C01854=1122.207,107.838,-57.449,-179.830,8.137,149.506
C01855=1122.202,108.087,-57.468,-179.828,8.140,149.507
C01856=1122.197,108.336,-57.487,-179.826,8.144,149.507
C01857=1122.193,108.586,-57.507,-179.823,8.148,149.507
C01858=1122.187,108.834,-57.526,-179.821,8.151,149.507
C01859=1122.183,109.084,-57.546,-179.818,8.156,149.507
C01860=1122.179,109.333,-57.565,-179.817,8.160,149.508
C01861=1122.173,109.582,-57.584,-179.815,8.163,149.508
C01862=1122.168,109.832,-57.604,-179.812,8.167,149.508
C01863=1122.163,110.081,-57.623,-179.810,8.171,149.509
C01864=1122.158,110.330,-57.642,-179.807,8.175,149.509
C01865=1122.154,110.579,-57.662,-179.805,8.179,149.509
C01866=1122.149,110.828,-57.681,-179.802,8.183,149.509
C01867=1122.144,111.078,-57.700,-179.800,8.186,149.509
C01868=1122.140,111.327,-57.720,-179.798,8.190,149.510
C01869=1122.135,111.576,-57.740,-179.796,8.193,149.510
C01870=1122.130,111.825,-57.760,-179.795,8.196,149.510
C01871=1122.125,112.075,-57.779,-179.793,8.200,149.511
C01872=1122.120,112.323,-57.798,-179.791,8.203,149.511
C01873=1122.116,112.573,-57.818,-179.789,8.207,149.511
C01874=1122.111,112.822,-57.838,-179.787,8.210,149.511
C01875=1122.106,113.071,-57.857,-179.786,8.214,149.512
C01876=1122.101,113.320,-57.877,-179.783,8.218,149.512
C01877=1122.096,113.570,-57.897,-179.781,8.221,149.512
C01878=1122.091,113.818,-57.917,-179.779,8.225,149.512
C01879=1122.087,114.068,-57.936,-179.778,8.228,149.513
C01880=1122.082,114.317,-57.956,-179.776,8.231,149.513
C01881=1122.077,114.567,-57.976,-179.774,8.235,149.513
C01882=1122.072,114.815,-57.996,-179.772,8.238,149.513
C01883=1122.067,115.065,-58.015,-179.771,8.242,149.514
C01884=1122.063,115.314,-58.035,-179.768,8.246,149.514
C01885=1122.058,115.563,-58.055,-179.766,8.249,149.514
C01886=1122.053,115.812,-58.075,-179.765,8.252,149.515
C01887=1122.048,116.062,-58.094,-179.763,8.256,149.515
C01888=1122.045,116.275,-58.111,-179.762,8.259,149.515
C01889=1122.041,116.490,-58.128,-179.760,8.262,149.515
C01890=1122.036,116.704,-58.146,-179.758,8.265,149.516
C01891=1122.032,116.919,-58.163,-179.757,8.268,149.516
C01892=1122.028,117.133,-58.180,-179.755,8.271,149.516
C01893=1122.024,117.347,-58.197,-179.753,8.274,149.516
C01894=1122.020,117.562,-58.214,-179.752,8.277,149.517
C01895=1122.015,117.776,-58.231,-179.751,8.279,149.517
C01896=1122.011,118.026,-58.251,-179.749,8.283,149.517
C01897=1122.006,118.275,-58.271,-179.746,8.286,149.517
C01898=1122.001,118.524,-58.291,-179.745,8.290,149.518
C01899=1121.996,118.773,-58.311,-179.743,8.294,149.518
C01900=1121.992,119.022,-58.331,-179.741,8.296,149.518
C01901=1121.987,119.271,-58.351,-179.739,8.300,149.518
C01902=1121.983,119.521,-58.371,-179.738,8.304,149.519
C01903=1121.978,119.770,-58.391,-179.736,8.307,149.519
C01904=1121.973,120.019,-58.411,-179.734,8.310,149.519
C01905=1121.968,120.267,-58.431,-179.732,8.313,149.519
C01906=1121.963,120.517,-58.452,-179.730,8.317,149.520
C01907=1121.958,120.766,-58.471,-179.728,8.321,149.520
C01908=1121.954,121.015,-58.492,-179.727,8.324,149.520
C01909=1121.949,121.265,-58.511,-179.725,8.327,149.520
C01910=1121.945,121.514,-58.532,-179.723,8.331,149.521
C01911=1121.940,121.763,-58.552,-179.721,8.334,149.521
C01912=1121.935,122.012,-58.571,-179.720,8.337,149.521
C01913=1121.930,122.261,-58.592,-179.718,8.341,149.522
C01914=1121.925,122.510,-58.612,-179.716,8.344,149.522
C01915=1121.921,122.759,-58.632,-179.714,8.348,149.522
C01916=1121.916,123.008,-58.653,-179.713,8.351,149.522
C01917=1121.912,123.257,-58.673,-179.711,8.354,149.523
C01918=1121.906,123.507,-58.693,-179.708,8.358,149.523
C01919=1121.902,123.756,-58.714,-179.706,8.361,149.523
C01920=1121.897,124.005,-58.734,-179.705,8.364,149.523
C01921=1121.893,124.255,-58.754,-179.703,8.368,149.524
C01922=1121.887,124.504,-58.775,-179.701,8.371,149.524
C01923=1121.882,124.752,-58.795,-179.700,8.374,149.524
C01924=1121.878,125.001,-58.815,-179.698,8.377,149.524
C01925=1121.873,125.251,-58.835,-179.696,8.381,149.525
C01926=1121.868,125.500,-58.856,-179.695,8.384,149.525
C01927=1121.864,125.749,-58.876,-179.693,8.388,149.525
C01928=1121.859,125.998,-58.897,-179.691,8.391,149.526
C01929=1121.855,126.247,-58.917,-179.689,8.395,149.526
C01930=1121.850,126.496,-58.938,-179.687,8.398,149.526
C01931=1121.845,126.746,-58.958,-179.685,8.401,149.526
C01932=1121.840,126.994,-58.978,-179.683,8.405,149.527
C01933=1121.835,127.244,-58.999,-179.682,8.407,149.527
C01934=1121.831,127.493,-59.019,-179.680,8.411,149.527
C01935=1121.826,127.742,-59.040,-179.678,8.415,149.528
C01936=1121.821,127.991,-59.061,-179.677,8.417,149.528
C01937=1121.817,128.240,-59.081,-179.675,8.421,149.528
C01938=1121.812,128.489,-59.101,-179.673,8.425,149.528
C01939=1121.807,128.739,-59.122,-179.672,8.428,149.529
C01940=1121.802,128.988,-59.142,-179.670,8.431,149.529
C01941=1121.797,129.237,-59.163,-179.668,8.435,149.529
C01942=1121.793,129.486,-59.183,-179.666,8.438,149.530
C01943=1121.788,129.735,-59.204,-179.664,8.441,149.530
C01944=1121.784,129.950,-59.222,-179.663,8.444,149.530
C01945=1121.780,130.163,-59.239,-179.662,8.447,149.530
C01946=1121.776,130.378,-59.257,-179.660,8.449,149.530
C01947=1121.772,130.592,-59.275,-179.659,8.452,149.531
C01948=1121.768,130.806,-59.292,-179.657,8.456,149.531
C01949=1121.764,131.021,-59.311,-179.656,8.459,149.531
C01950=1121.759,131.235,-59.328,-179.654,8.461,149.532
C01951=1121.756,131.449,-59.346,-179.653,8.464,149.532
C01952=1121.751,131.699,-59.367,-179.651,8.467,149.532
C01953=1121.746,131.947,-59.387,-179.650,8.471,149.532
C01954=1121.741,132.196,-59.409,-179.648,8.474,149.533
C01955=1121.737,132.445,-59.429,-179.646,8.477,149.533
C01956=1121.732,132.694,-59.450,-179.644,8.480,149.533
C01957=1121.727,132.943,-59.471,-179.642,8.484,149.534
C01958=1121.722,133.193,-59.492,-179.641,8.487,149.534
C01959=1121.718,133.441,-59.512,-179.639,8.490,149.534
C01960=1121.713,133.691,-59.533,-179.638,8.493,149.534
C01961=1121.709,133.940,-59.554,-179.636,8.497,149.535
C01962=1121.704,134.189,-59.575,-179.634,8.500,149.535
C01963=1121.699,134.438,-59.596,-179.633,8.504,149.535
C01964=1121.694,134.687,-59.617,-179.631,8.507,149.536
C01965=1121.690,134.936,-59.637,-179.629,8.510,149.536
C01966=1121.685,135.185,-59.658,-179.628,8.514,149.536
C01967=1121.680,135.434,-59.679,-179.625,8.517,149.536
C01968=1121.675,135.683,-59.700,-179.624,8.520,149.537
C01969=1121.671,135.933,-59.721,-179.622,8.524,149.537
C01970=1121.666,136.182,-59.742,-179.621,8.526,149.537
C01971=1121.661,136.431,-59.764,-179.619,8.530,149.538
C01972=1121.657,136.680,-59.784,-179.617,8.534,149.538
C01973=1121.652,136.929,-59.805,-179.616,8.536,149.538
C01974=1121.647,137.178,-59.826,-179.614,8.540,149.539
C01975=1121.643,137.426,-59.847,-179.613,8.543,149.539
C01976=1121.638,137.676,-59.868,-179.611,8.547,149.539
C01977=1121.633,137.926,-59.889,-179.609,8.550,149.540
C01978=1121.629,138.174,-59.910,-179.608,8.554,149.540
C01979=1121.623,138.423,-59.931,-179.606,8.557,149.540
C01980=1121.619,138.672,-59.952,-179.604,8.560,149.540
C01981=1121.615,138.921,-59.974,-179.603,8.564,149.541
C01982=1121.610,139.171,-59.995,-179.601,8.566,149.541
C01983=1121.605,139.419,-60.016,-179.600,8.570,149.542
C01984=1121.600,139.668,-60.037,-179.598,8.574,149.542
C01985=1121.595,139.918,-60.058,-179.597,8.577,149.542
C01986=1121.591,140.167,-60.080,-179.595,8.580,149.542
C01987=1121.586,140.416,-60.100,-179.594,8.583,149.543
C01988=1121.582,140.665,-60.122,-179.592,8.587,149.543
C01989=1121.576,140.914,-60.143,-179.591,8.590,149.544
C01990=1121.573,141.163,-60.164,-179.588,8.593,149.544
C01991=1121.568,141.412,-60.185,-179.587,8.596,149.544
C01992=1121.563,141.661,-60.207,-179.585,8.600,149.544
C01993=1121.558,141.910,-60.228,-179.584,8.604,149.545
C01994=1121.554,142.159,-60.249,-179.582,8.607,149.545
C01995=1121.549,142.408,-60.270,-179.581,8.610,149.546
C01996=1121.544,142.657,-60.292,-179.579,8.613,149.546
C01997=1121.539,142.906,-60.313,-179.578,8.617,149.546
C01998=1121.535,143.155,-60.334,-179.576,8.620,149.546
C01999=1121.530,143.404,-60.355,-179.574,8.624,149.547
C02000=1121.526,143.619,-60.374,-179.573,8.626,149.547
C02001=1121.522,143.832,-60.392,-179.572,8.629,149.548
C02002=1121.518,144.047,-60.411,-179.571,8.632,149.548
C02003=1121.514,144.261,-60.429,-179.569,8.635,149.548
C02004=1121.510,144.475,-60.448,-179.568,8.638,149.548
C02005=1121.506,144.690,-60.466,-179.567,8.641,149.549
C02006=1121.502,144.903,-60.484,-179.565,8.643,149.549
C02007=1121.497,145.118,-60.503,-179.564,8.646,149.549
C02008=1121.493,145.366,-60.524,-179.561,8.651,149.550
C02009=1121.489,145.616,-60.546,-179.559,8.654,149.550
C02010=1121.484,145.865,-60.567,-179.557,8.658,149.550
C02011=1121.479,146.114,-60.588,-179.555,8.662,149.550
C02012=1121.475,146.363,-60.610,-179.552,8.666,149.550
C02013=1121.469,146.612,-60.631,-179.549,8.669,149.551
C02014=1121.464,146.861,-60.653,-179.547,8.674,149.551
C02015=1121.460,147.110,-60.675,-179.545,8.677,149.551
C02016=1121.455,147.359,-60.697,-179.542,8.681,149.551
C02017=1121.451,147.609,-60.718,-179.540,8.685,149.551
C02018=1121.447,147.857,-60.739,-179.538,8.688,149.552
C02019=1121.442,148.106,-60.761,-179.535,8.693,149.552
C02020=1121.438,148.355,-60.783,-179.533,8.696,149.552
C02021=1121.433,148.604,-60.805,-179.530,8.700,149.552
C02022=1121.427,148.853,-60.826,-179.528,8.703,149.552
C02023=1121.423,149.102,-60.848,-179.526,8.707,149.553
C02024=1121.418,149.351,-60.869,-179.523,8.711,149.553
C02025=1121.414,149.600,-60.891,-179.520,8.714,149.553
C02026=1121.409,149.849,-60.913,-179.518,8.719,149.553
C02027=1121.404,150.098,-60.935,-179.516,8.722,149.553
C02028=1121.400,150.347,-60.957,-179.513,8.726,149.554
C02029=1121.394,150.596,-60.979,-179.510,8.729,149.554
C02030=1121.390,150.845,-61.001,-179.508,8.733,149.554
C02031=1121.385,151.094,-61.023,-179.506,8.736,149.554
C02032=1121.381,151.343,-61.045,-179.504,8.740,149.554
C02033=1121.376,151.592,-61.067,-179.501,8.744,149.554
C02034=1121.372,151.842,-61.088,-179.499,8.747,149.555
C02035=1121.367,152.090,-61.110,-179.497,8.751,149.555
C02036=1121.362,152.338,-61.132,-179.494,8.755,149.555
C02037=1121.358,152.588,-61.154,-179.492,8.758,149.555
C02038=1121.353,152.836,-61.176,-179.489,8.762,149.555
C02039=1121.348,153.086,-61.198,-179.487,8.765,149.555
C02040=1121.343,153.335,-61.220,-179.484,8.769,149.556
C02041=1121.339,153.584,-61.242,-179.482,8.772,149.556
C02042=1121.334,153.833,-61.264,-179.480,8.776,149.556
C02043=1121.330,154.082,-61.286,-179.478,8.779,149.556
C02044=1121.325,154.331,-61.307,-179.475,8.782,149.556
C02045=1121.320,154.580,-61.330,-179.472,8.786,149.556
C02046=1121.316,154.830,-61.352,-179.470,8.790,149.556
C02047=1121.311,155.078,-61.375,-179.468,8.793,149.557
C02048=1121.307,155.327,-61.397,-179.465,8.796,149.557
C02049=1121.302,155.576,-61.418,-179.463,8.800,149.557
C02050=1121.297,155.825,-61.441,-179.461,8.803,149.557
C02051=1121.292,156.074,-61.463,-179.458,8.807,149.557
C02052=1121.288,156.323,-61.485,-179.455,8.810,149.557
C02053=1121.283,156.571,-61.507,-179.453,8.814,149.557
C02054=1121.278,156.821,-61.530,-179.451,8.817,149.558
C02055=1121.274,157.070,-61.552,-179.449,8.820,149.558
C02056=1121.270,157.284,-61.572,-179.446,8.823,149.558
C02057=1121.266,157.498,-61.591,-179.445,8.826,149.558
C02058=1121.262,157.712,-61.610,-179.442,8.829,149.558
C02059=1121.258,157.927,-61.629,-179.441,8.832,149.558
C02060=1121.254,158.141,-61.648,-179.438,8.835,149.558
C02061=1121.250,158.355,-61.667,-179.436,8.837,149.558
C02062=1121.247,158.568,-61.686,-179.434,8.841,149.559
C02063=1121.243,158.782,-61.705,-179.432,8.843,149.559
C02064=1121.237,159.031,-61.728,-179.430,8.847,149.559
C02065=1121.233,159.280,-61.750,-179.428,8.850,149.559
C02066=1121.229,159.529,-61.772,-179.426,8.853,149.559
C02067=1121.223,159.778,-61.795,-179.423,8.856,149.559
C02068=1121.219,160.027,-61.817,-179.421,8.859,149.559
C02069=1121.214,160.277,-61.840,-179.418,8.864,149.559
C02070=1121.210,160.525,-61.862,-179.415,8.867,149.559
C02071=1121.205,160.774,-61.885,-179.413,8.870,149.560
C02072=1121.201,161.023,-61.908,-179.411,8.873,149.560
C02073=1121.196,161.272,-61.930,-179.408,8.876,149.560
C02074=1121.191,161.521,-61.953,-179.406,8.880,149.560
C02075=1121.187,161.770,-61.975,-179.404,8.882,149.560
C02076=1121.182,162.018,-61.997,-179.402,8.885,149.560
C02077=1121.177,162.268,-62.020,-179.400,8.889,149.560
C02078=1121.173,162.516,-62.043,-179.397,8.892,149.560
C02079=1121.168,162.765,-62.065,-179.395,8.895,149.561
C02080=1121.164,163.014,-62.088,-179.393,8.899,149.561
C02081=1121.159,163.263,-62.111,-179.390,8.902,149.561
C02082=1121.155,163.513,-62.133,-179.388,8.905,149.561
C02083=1121.149,163.761,-62.156,-179.385,8.908,149.561
C02084=1121.145,164.010,-62.178,-179.383,8.911,149.561
C02085=1121.141,164.259,-62.202,-179.381,8.915,149.561
C02086=1121.137,164.508,-62.224,-179.378,8.918,149.561
C02087=1121.131,164.757,-62.247,-179.376,8.921,149.561
C02088=1121.127,165.006,-62.269,-179.374,8.925,149.561
C02089=1121.122,165.255,-62.293,-179.371,8.928,149.561
C02090=1121.118,165.504,-62.315,-179.369,8.930,149.562
C02091=1121.113,165.752,-62.338,-179.367,8.933,149.562
C02092=1121.108,166.001,-62.361,-179.365,8.937,149.562
C02093=1121.104,166.250,-62.384,-179.362,8.940,149.562
C02094=1121.099,166.500,-62.407,-179.360,8.943,149.562
C02095=1121.095,166.748,-62.429,-179.357,8.946,149.562
C02096=1121.090,166.997,-62.452,-179.355,8.949,149.562
C02097=1121.085,167.246,-62.476,-179.353,8.952,149.562
C02098=1121.081,167.495,-62.498,-179.351,8.955,149.562
C02099=1121.076,167.744,-62.521,-179.348,8.958,149.562
C02100=1121.071,167.993,-62.544,-179.346,8.961,149.562
C02101=1121.067,168.241,-62.567,-179.344,8.965,149.563
C02102=1121.062,168.490,-62.590,-179.341,8.968,149.563
C02103=1121.057,168.739,-62.614,-179.339,8.970,149.563
C02104=1121.053,168.988,-62.636,-179.337,8.974,149.563
C02105=1121.048,169.238,-62.659,-179.335,8.977,149.563
C02106=1121.044,169.487,-62.682,-179.332,8.980,149.563
C02107=1121.039,169.735,-62.705,-179.330,8.983,149.563
C02108=1121.035,169.984,-62.728,-179.328,8.986,149.563
C02109=1121.030,170.233,-62.751,-179.326,8.989,149.563
C02110=1121.026,170.482,-62.774,-179.323,8.992,149.563
C02111=1121.021,170.731,-62.798,-179.321,8.996,149.564
C02112=1121.017,170.944,-62.817,-179.319,8.998,149.564
C02113=1121.013,171.158,-62.838,-179.317,9.000,149.564
C02114=1121.009,171.373,-62.857,-179.315,9.003,149.564
C02115=1121.006,171.586,-62.877,-179.313,9.006,149.564
C02116=1121.001,171.800,-62.897,-179.312,9.008,149.564
C02117=1120.997,172.014,-62.917,-179.310,9.011,149.564
C02118=1120.994,172.229,-62.937,-179.308,9.013,149.564
C02119=1120.989,172.443,-62.957,-179.306,9.016,149.564
C02120=1120.985,172.692,-62.980,-179.304,9.019,149.564
C02121=1120.981,172.940,-63.003,-179.301,9.022,149.564
C02122=1120.976,173.189,-63.027,-179.300,9.025,149.565
C02123=1120.971,173.437,-63.050,-179.297,9.028,149.565
C02124=1120.966,173.686,-63.074,-179.295,9.031,149.565
C02125=1120.962,173.935,-63.097,-179.292,9.034,149.565
C02126=1120.957,174.184,-63.120,-179.291,9.037,149.565
C02127=1120.953,174.433,-63.143,-179.288,9.040,149.565
C02128=1120.948,174.682,-63.167,-179.286,9.043,149.565
C02129=1120.943,174.931,-63.190,-179.284,9.046,149.565
C02130=1120.939,175.179,-63.214,-179.282,9.049,149.565
C02131=1120.934,175.428,-63.237,-179.279,9.052,149.565
C02132=1120.930,175.677,-63.261,-179.278,9.055,149.566
C02133=1120.925,175.927,-63.284,-179.275,9.058,149.566
C02134=1120.921,176.175,-63.307,-179.273,9.061,149.566
C02135=1120.917,176.424,-63.331,-179.271,9.063,149.566
C02136=1120.912,176.673,-63.354,-179.269,9.067,149.566
C02137=1120.907,176.922,-63.378,-179.266,9.070,149.566
C02138=1120.903,177.171,-63.401,-179.264,9.072,149.566
C02139=1120.898,177.419,-63.425,-179.262,9.075,149.566
C02140=1120.893,177.668,-63.448,-179.260,9.079,149.566
C02141=1120.889,177.917,-63.472,-179.258,9.081,149.566
C02142=1120.884,178.166,-63.496,-179.256,9.084,149.567
C02143=1120.880,178.415,-63.519,-179.254,9.087,149.567
C02144=1120.875,178.664,-63.543,-179.252,9.090,149.567
C02145=1120.871,178.912,-63.567,-179.249,9.093,149.567
C02146=1120.866,179.161,-63.590,-179.247,9.096,149.567
C02147=1120.861,179.410,-63.613,-179.245,9.099,149.567
C02148=1120.857,179.659,-63.637,-179.242,9.103,149.567
C02149=1120.852,179.908,-63.661,-179.239,9.106,149.567
C02150=1120.848,180.157,-63.684,-179.237,9.109,149.567
C02151=1120.844,180.406,-63.709,-179.234,9.112,149.567
C02152=1120.839,180.655,-63.732,-179.231,9.116,149.567
C02153=1120.834,180.903,-63.756,-179.228,9.119,149.567
C02154=1120.830,181.152,-63.779,-179.225,9.122,149.567
C02155=1120.825,181.401,-63.803,-179.223,9.125,149.567
C02156=1120.821,181.650,-63.827,-179.220,9.128,149.567
C02157=1120.816,181.898,-63.851,-179.218,9.131,149.567
C02158=1120.812,182.147,-63.874,-179.215,9.135,149.567
C02159=1120.807,182.396,-63.898,-179.212,9.138,149.567
C02160=1120.802,182.646,-63.923,-179.209,9.141,149.567
C02161=1120.798,182.894,-63.947,-179.207,9.144,149.567
C02162=1120.793,183.143,-63.970,-179.204,9.147,149.567
C02163=1120.789,183.391,-63.994,-179.202,9.150,149.567
C02164=1120.784,183.640,-64.018,-179.199,9.153,149.567
C02165=1120.780,183.889,-64.042,-179.197,9.156,149.567
C02166=1120.775,184.137,-64.066,-179.194,9.159,149.567
C02167=1120.771,184.387,-64.091,-179.191,9.162,149.567
C02168=1120.767,184.600,-64.110,-179.189,9.164,149.567
C02169=1120.763,184.814,-64.131,-179.187,9.167,149.567
C02170=1120.759,185.028,-64.152,-179.185,9.170,149.567
C02171=1120.755,185.242,-64.172,-179.183,9.172,149.567
C02172=1120.751,185.456,-64.193,-179.181,9.175,149.567
C02173=1120.747,185.670,-64.214,-179.179,9.177,149.567
C02174=1120.744,185.884,-64.234,-179.177,9.180,149.568
C02175=1120.740,186.097,-64.255,-179.175,9.182,149.568
C02176=1120.735,186.346,-64.279,-179.172,9.185,149.567
C02177=1120.730,186.596,-64.304,-179.170,9.187,149.567
C02178=1120.726,186.844,-64.328,-179.167,9.191,149.567
C02179=1120.722,187.092,-64.352,-179.165,9.194,149.568
C02180=1120.717,187.341,-64.376,-179.162,9.197,149.568
C02181=1120.712,187.591,-64.400,-179.160,9.199,149.568
C02182=1120.708,187.839,-64.424,-179.158,9.202,149.568
C02183=1120.704,188.088,-64.448,-179.155,9.205,149.568
C02184=1120.698,188.336,-64.473,-179.153,9.208,149.568
C02185=1120.694,188.585,-64.497,-179.151,9.211,149.568
C02186=1120.690,188.834,-64.522,-179.149,9.213,149.568
C02187=1120.685,189.083,-64.546,-179.146,9.216,149.568
C02188=1120.680,189.332,-64.570,-179.144,9.219,149.568
C02189=1120.676,189.580,-64.594,-179.142,9.222,149.568
C02190=1120.672,189.829,-64.619,-179.140,9.225,149.568
C02191=1120.667,190.078,-64.643,-179.138,9.227,149.568
C02192=1120.662,190.327,-64.667,-179.135,9.230,149.568
C02193=1120.658,190.576,-64.692,-179.133,9.232,149.568
C02194=1120.654,190.824,-64.716,-179.131,9.236,149.568
C02195=1120.649,191.073,-64.741,-179.129,9.238,149.568
C02196=1120.644,191.321,-64.765,-179.127,9.241,149.568
C02197=1120.640,191.571,-64.790,-179.125,9.244,149.568
C02198=1120.635,191.819,-64.814,-179.123,9.246,149.569
C02199=1120.631,192.067,-64.838,-179.120,9.249,149.569
C02200=1120.626,192.317,-64.863,-179.119,9.252,149.569
C02201=1120.622,192.565,-64.887,-179.117,9.254,149.569
C02202=1120.617,192.814,-64.912,-179.115,9.257,149.569
C02203=1120.613,193.063,-64.936,-179.113,9.260,149.569
C02204=1120.608,193.312,-64.961,-179.111,9.262,149.569
C02205=1120.604,193.560,-64.985,-179.109,9.265,149.569
C02206=1120.599,193.810,-65.010,-179.107,9.268,149.569
C02207=1120.595,194.058,-65.034,-179.105,9.270,149.569
C02208=1120.590,194.307,-65.059,-179.103,9.273,149.570
C02209=1120.586,194.556,-65.083,-179.101,9.276,149.570
C02210=1120.581,194.805,-65.108,-179.099,9.279,149.570
C02211=1120.577,195.052,-65.133,-179.097,9.281,149.570
C02212=1120.572,195.302,-65.158,-179.096,9.284,149.570
C02213=1120.568,195.550,-65.182,-179.094,9.286,149.570
C02214=1120.563,195.800,-65.207,-179.092,9.289,149.570
C02215=1120.559,196.048,-65.231,-179.090,9.292,149.570
C02216=1120.554,196.297,-65.255,-179.089,9.295,149.571
C02217=1120.550,196.545,-65.281,-179.086,9.298,149.571
C02218=1120.545,196.794,-65.305,-179.083,9.301,149.571
C02219=1120.541,197.043,-65.330,-179.079,9.305,149.570
C02220=1120.536,197.292,-65.354,-179.076,9.309,149.570
C02221=1120.532,197.540,-65.379,-179.072,9.312,149.570
C02222=1120.527,197.789,-65.404,-179.069,9.315,149.570
C02223=1120.522,198.038,-65.429,-179.066,9.319,149.570
C02224=1120.519,198.252,-65.450,-179.063,9.321,149.570
C02225=1120.515,198.466,-65.472,-179.061,9.325,149.570
C02226=1120.511,198.679,-65.493,-179.058,9.327,149.570
C02227=1120.507,198.893,-65.514,-179.055,9.330,149.570
C02228=1120.504,199.107,-65.536,-179.052,9.333,149.570
C02229=1120.499,199.320,-65.557,-179.049,9.336,149.570
C02230=1120.496,199.534,-65.578,-179.046,9.339,149.570
C02231=1120.492,199.748,-65.600,-179.044,9.342,149.570
C02232=1120.487,199.997,-65.625,-179.041,9.344,149.570
C02233=1120.484,200.245,-65.650,-179.037,9.348,149.569
C02234=1120.478,200.494,-65.674,-179.034,9.351,149.569
C02235=1120.474,200.743,-65.700,-179.031,9.355,149.569
C02236=1120.469,200.992,-65.725,-179.028,9.357,149.569
C02237=1120.466,201.240,-65.750,-179.025,9.360,149.569
C02238=1120.460,201.489,-65.775,-179.022,9.364,149.569
C02239=1120.456,201.738,-65.800,-179.019,9.366,149.569
C02240=1120.451,201.986,-65.825,-179.016,9.369,149.569
C02241=1120.448,202.235,-65.850,-179.013,9.373,149.569
C02242=1120.443,202.484,-65.875,-179.010,9.376,149.569
C02243=1120.438,202.732,-65.901,-179.007,9.378,149.568
C02244=1120.433,202.980,-65.926,-179.004,9.381,149.568
C02245=1120.430,203.230,-65.950,-179.001,9.385,149.568
C02246=1120.425,203.478,-65.976,-178.998,9.388,149.568
C02247=1120.420,203.727,-66.001,-178.995,9.391,149.568
C02248=1120.416,203.976,-66.027,-178.992,9.393,149.568
C02249=1120.411,204.224,-66.052,-178.989,9.396,149.568
C02250=1120.407,204.473,-66.077,-178.986,9.399,149.568
C02251=1120.403,204.722,-66.103,-178.983,9.402,149.568
C02252=1120.398,204.970,-66.128,-178.980,9.405,149.567
C02253=1120.394,205.219,-66.153,-178.977,9.408,149.567
C02254=1120.389,205.468,-66.178,-178.974,9.411,149.567
C02255=1120.385,205.716,-66.204,-178.971,9.414,149.567
C02256=1120.381,205.965,-66.230,-178.968,9.417,149.567
C02257=1120.375,206.214,-66.254,-178.966,9.420,149.567
C02258=1120.371,206.463,-66.280,-178.963,9.423,149.567
C02259=1120.366,206.711,-66.305,-178.961,9.425,149.567
C02260=1120.362,206.960,-66.331,-178.958,9.428,149.567
C02261=1120.358,207.208,-66.357,-178.955,9.430,149.567
C02262=1120.353,207.457,-66.382,-178.952,9.433,149.567
C02263=1120.349,207.706,-66.407,-178.950,9.436,149.567
C02264=1120.344,207.955,-66.433,-178.947,9.439,149.567
C02265=1120.340,208.203,-66.458,-178.944,9.442,149.567
C02266=1120.335,208.452,-66.484,-178.941,9.445,149.566
C02267=1120.331,208.700,-66.510,-178.939,9.448,149.566
C02268=1120.326,208.949,-66.535,-178.936,9.450,149.566
C02269=1120.322,209.197,-66.561,-178.934,9.453,149.566
C02270=1120.318,209.446,-66.587,-178.931,9.456,149.566
C02271=1120.314,209.695,-66.613,-178.928,9.459,149.566
C02272=1120.309,209.943,-66.638,-178.926,9.462,149.566
C02273=1120.305,210.192,-66.664,-178.923,9.464,149.566
C02274=1120.300,210.441,-66.689,-178.921,9.467,149.566
C02275=1120.296,210.689,-66.715,-178.918,9.470,149.566
C02276=1120.291,210.938,-66.741,-178.916,9.473,149.566
C02277=1120.287,211.186,-66.766,-178.914,9.475,149.566
C02278=1120.282,211.436,-66.793,-178.911,9.478,149.566
C02279=1120.277,211.684,-66.818,-178.909,9.481,149.566
C02280=1120.274,211.898,-66.840,-178.907,9.484,149.566
C02281=1120.270,212.111,-66.862,-178.905,9.486,149.566
C02282=1120.266,212.325,-66.885,-178.903,9.488,149.566
C02283=1120.263,212.539,-66.906,-178.901,9.491,149.567
C02284=1120.259,212.752,-66.929,-178.898,9.494,149.567
C02285=1120.255,212.966,-66.951,-178.897,9.496,149.567
C02286=1120.251,213.180,-66.973,-178.895,9.499,149.567
C02287=1120.248,213.393,-66.995,-178.893,9.501,149.567
C02288=1120.242,213.642,-67.021,-178.891,9.504,149.567
C02289=1120.238,213.890,-67.047,-178.889,9.507,149.567
C02290=1120.234,214.139,-67.073,-178.887,9.509,149.567
C02291=1120.230,214.387,-67.099,-178.885,9.513,149.567
C02292=1120.226,214.636,-67.125,-178.883,9.515,149.567
C02293=1120.221,214.884,-67.150,-178.881,9.518,149.568
C02294=1120.216,215.133,-67.177,-178.879,9.521,149.568
C02295=1120.212,215.382,-67.202,-178.876,9.524,149.568
C02296=1120.208,215.630,-67.229,-178.875,9.526,149.568
C02297=1120.203,215.879,-67.255,-178.872,9.530,149.568
C02298=1120.198,216.128,-67.281,-178.870,9.532,149.568
C02299=1120.194,216.376,-67.306,-178.868,9.535,149.568
C02300=1120.190,216.625,-67.333,-178.866,9.538,149.568
C02301=1120.185,216.873,-67.359,-178.864,9.541,149.568
C02302=1120.181,217.122,-67.385,-178.862,9.544,149.569
C02303=1120.177,217.371,-67.411,-178.859,9.547,149.569
C02304=1120.170,217.694,-67.445,-178.857,9.551,149.569
C02305=1120.165,218.019,-67.479,-178.854,9.555,149.569
C02306=1120.159,218.343,-67.513,-178.851,9.559,149.569
C02307=1120.154,218.667,-67.548,-178.848,9.563,149.569
C02308=1120.149,218.915,-67.573,-178.845,9.566,149.569
C02309=1120.144,219.164,-67.600,-178.843,9.569,149.570
C02310=1120.140,219.412,-67.626,-178.841,9.572,149.570
C02311=1120.136,219.661,-67.651,-178.838,9.575,149.570
C02312=1120.131,219.910,-67.679,-178.836,9.578,149.570
C02313=1120.127,220.158,-67.704,-178.833,9.582,149.570
C02314=1120.122,220.407,-67.731,-178.831,9.584,149.570
C02315=1120.118,220.656,-67.757,-178.829,9.587,149.570
C02316=1120.114,220.904,-67.784,-178.826,9.590,149.570
C02317=1120.109,221.153,-67.810,-178.824,9.594,149.570
C02318=1120.105,221.401,-67.836,-178.821,9.597,149.570
C02319=1120.101,221.650,-67.863,-178.819,9.600,149.570
C02320=1120.096,221.898,-67.889,-178.816,9.603,149.571
C02321=1120.091,222.147,-67.915,-178.813,9.607,149.571
C02322=1120.087,222.395,-67.942,-178.811,9.610,149.571
C02323=1120.083,222.643,-67.968,-178.808,9.613,149.571
C02324=1120.078,222.892,-67.994,-178.805,9.616,149.571
C02325=1120.074,223.141,-68.021,-178.803,9.619,149.571
C02326=1120.069,223.390,-68.047,-178.800,9.622,149.571
C02327=1120.065,223.638,-68.074,-178.798,9.625,149.571
C02328=1120.061,223.886,-68.101,-178.794,9.629,149.571
C02329=1120.057,224.135,-68.127,-178.792,9.632,149.571
C02330=1120.052,224.384,-68.154,-178.789,9.635,149.571
C02331=1120.048,224.632,-68.180,-178.786,9.638,149.571
C02332=1120.043,224.880,-68.207,-178.784,9.641,149.571
C02333=1120.039,225.129,-68.233,-178.781,9.645,149.571
C02334=1120.034,225.378,-68.260,-178.778,9.648,149.571
C02335=1120.030,225.626,-68.287,-178.775,9.651,149.571
C02336=1120.024,225.979,-68.325,-178.772,9.655,149.571
C02337=1120.018,226.330,-68.363,-178.767,9.661,149.571
C02338=1120.012,226.682,-68.400,-178.762,9.665,149.571
C02339=1120.005,227.033,-68.438,-178.759,9.669,149.571
C02340=1120.002,227.281,-68.465,-178.756,9.672,149.571
C02341=1119.997,227.530,-68.491,-178.753,9.676,149.571
C02342=1119.992,227.779,-68.518,-178.750,9.679,149.571
C02343=1119.988,228.027,-68.544,-178.746,9.682,149.571
C02344=1119.983,228.275,-68.572,-178.743,9.685,149.571
C02345=1119.979,228.524,-68.599,-178.741,9.688,149.571
C02346=1119.975,228.773,-68.625,-178.737,9.692,149.571
C02347=1119.971,229.021,-68.652,-178.734,9.695,149.570
C02348=1119.966,229.270,-68.680,-178.731,9.698,149.571
C02349=1119.961,229.518,-68.707,-178.728,9.701,149.570
C02350=1119.957,229.766,-68.733,-178.724,9.705,149.570
C02351=1119.953,230.015,-68.760,-178.721,9.707,149.570
C02352=1119.948,230.263,-68.787,-178.718,9.711,149.570
C02353=1119.944,230.513,-68.815,-178.714,9.714,149.570
C02354=1119.940,230.761,-68.841,-178.711,9.717,149.570
C02355=1119.936,231.009,-68.868,-178.708,9.720,149.570
C02356=1119.931,231.258,-68.895,-178.705,9.723,149.570
C02357=1119.926,231.506,-68.922,-178.702,9.726,149.569
C02358=1119.922,231.754,-68.949,-178.699,9.729,149.569
C02359=1119.919,232.003,-68.977,-178.696,9.733,149.569
C02360=1119.914,232.251,-69.004,-178.693,9.736,149.569
C02361=1119.909,232.500,-69.031,-178.690,9.738,149.569
C02362=1119.905,232.748,-69.058,-178.687,9.741,149.569
C02363=1119.900,232.997,-69.085,-178.684,9.744,149.569
C02364=1119.896,233.246,-69.113,-178.681,9.747,149.569
C02365=1119.892,233.494,-69.140,-178.677,9.750,149.569
C02366=1119.888,233.742,-69.167,-178.674,9.753,149.569
C02367=1119.883,233.991,-69.194,-178.671,9.756,149.568
C02368=1119.879,234.239,-69.222,-178.669,9.758,149.568
C02369=1119.875,234.488,-69.249,-178.666,9.761,149.568
C02370=1119.870,234.736,-69.276,-178.663,9.764,149.568
C02371=1119.865,234.985,-69.303,-178.660,9.767,149.568
C02372=1119.861,235.233,-69.331,-178.657,9.770,149.568
C02373=1119.857,235.482,-69.358,-178.654,9.772,149.568
C02374=1119.852,235.730,-69.385,-178.652,9.774,149.568
C02375=1119.848,235.978,-69.413,-178.649,9.777,149.568
C02376=1119.844,236.227,-69.440,-178.646,9.780,149.567
C02377=1119.840,236.475,-69.468,-178.643,9.783,149.567
C02378=1119.835,236.723,-69.495,-178.640,9.785,149.567
C02379=1119.831,236.973,-69.522,-178.638,9.788,149.567
C02380=1119.827,237.221,-69.550,-178.635,9.791,149.567
C02381=1119.822,237.469,-69.577,-178.632,9.793,149.567
C02382=1119.819,237.718,-69.605,-178.629,9.796,149.567
C02383=1119.813,237.966,-69.633,-178.627,9.798,149.567
C02384=1119.809,238.214,-69.661,-178.625,9.801,149.567
C02385=1119.805,238.464,-69.688,-178.622,9.804,149.567
C02386=1119.801,238.711,-69.716,-178.619,9.806,149.567
C02387=1119.796,238.960,-69.743,-178.616,9.809,149.566
C02388=1119.793,239.174,-69.767,-178.614,9.811,149.566
C02389=1119.789,239.387,-69.790,-178.612,9.813,149.566
C02390=1119.785,239.600,-69.814,-178.610,9.815,149.566
C02391=1119.781,239.814,-69.838,-178.608,9.817,149.566
C02392=1119.778,240.027,-69.862,-178.606,9.820,149.566
C02393=1119.774,240.240,-69.885,-178.604,9.821,149.566
C02394=1119.771,240.453,-69.909,-178.602,9.824,149.566
C02395=1119.766,240.667,-69.933,-178.600,9.826,149.566
C02396=1119.762,240.915,-69.960,-178.598,9.828,149.566
C02397=1119.758,241.164,-69.989,-178.595,9.831,149.566
C02398=1119.754,241.412,-70.016,-178.593,9.833,149.566
C02399=1119.750,241.661,-70.044,-178.590,9.835,149.566
C02400=1119.745,241.909,-70.072,-178.588,9.838,149.566
C02401=1119.740,242.157,-70.100,-178.586,9.840,149.566
C02402=1119.736,242.406,-70.127,-178.584,9.843,149.566
C02403=1119.732,242.654,-70.155,-178.581,9.845,149.566
C02404=1119.728,242.903,-70.183,-178.579,9.848,149.566
C02405=1119.723,243.151,-70.210,-178.577,9.850,149.566
C02406=1119.719,243.399,-70.238,-178.575,9.852,149.566
C02407=1119.714,243.648,-70.267,-178.572,9.855,149.566
C02408=1119.710,243.896,-70.295,-178.570,9.857,149.566
C02409=1119.706,244.145,-70.322,-178.568,9.860,149.566
C02410=1119.702,244.393,-70.350,-178.566,9.862,149.566
C02411=1119.698,244.641,-70.378,-178.565,9.864,149.566
C02412=1119.693,244.890,-70.406,-178.563,9.867,149.566
C02413=1119.689,245.139,-70.434,-178.560,9.870,149.566
C02414=1119.684,245.387,-70.462,-178.558,9.872,149.566
C02415=1119.680,245.635,-70.489,-178.556,9.875,149.566
C02416=1119.676,245.883,-70.518,-178.554,9.877,149.566
C02417=1119.671,246.131,-70.546,-178.553,9.879,149.567
C02418=1119.667,246.380,-70.574,-178.551,9.882,149.567
C02419=1119.662,246.629,-70.602,-178.549,9.884,149.567
C02420=1119.658,246.877,-70.630,-178.547,9.886,149.567
C02421=1119.654,247.125,-70.658,-178.545,9.889,149.567
C02422=1119.650,247.374,-70.686,-178.544,9.891,149.567
C02423=1119.645,247.622,-70.714,-178.540,9.895,149.567
C02424=1119.641,247.871,-70.742,-178.535,9.899,149.567
C02425=1119.637,248.118,-70.770,-178.529,9.904,149.566
C02426=1119.633,248.367,-70.799,-178.524,9.908,149.566
C02427=1119.628,248.615,-70.826,-178.520,9.912,149.566
C02428=1119.624,248.864,-70.855,-178.515,9.916,149.565
C02429=1119.619,249.112,-70.883,-178.511,9.920,149.565
C02430=1119.616,249.360,-70.911,-178.505,9.923,149.565
C02431=1119.611,249.609,-70.940,-178.502,9.926,149.564
C02432=1119.607,249.857,-70.968,-178.497,9.930,149.564
C02433=1119.602,250.106,-70.996,-178.493,9.934,149.564
C02434=1119.598,250.354,-71.024,-178.489,9.937,149.563
C02435=1119.594,250.603,-71.052,-178.485,9.940,149.563
C02436=1119.590,250.851,-71.082,-178.482,9.943,149.563
C02437=1119.586,251.099,-71.110,-178.478,9.946,149.563
C02438=1119.581,251.348,-71.138,-178.475,9.948,149.562
C02439=1119.577,251.595,-71.166,-178.472,9.951,149.562
C02440=1119.572,251.844,-71.195,-178.468,9.953,149.562
C02441=1119.569,252.092,-71.224,-178.465,9.956,149.562
C02442=1119.564,252.341,-71.252,-178.462,9.959,149.562
C02443=1119.560,252.589,-71.280,-178.460,9.961,149.562
C02444=1119.556,252.803,-71.305,-178.458,9.963,149.562
C02445=1119.552,253.016,-71.329,-178.455,9.965,149.561
C02446=1119.549,253.229,-71.354,-178.453,9.967,149.561
C02447=1119.545,253.442,-71.378,-178.452,9.968,149.561
C02448=1119.541,253.656,-71.403,-178.450,9.970,149.561
C02449=1119.538,253.868,-71.428,-178.448,9.972,149.561
C02450=1119.534,254.082,-71.452,-178.446,9.974,149.561
C02451=1119.530,254.296,-71.477,-178.445,9.975,149.561
C02452=1119.526,254.543,-71.505,-178.444,9.977,149.561
C02453=1119.522,254.792,-71.534,-178.442,9.979,149.561
C02454=1119.518,255.040,-71.563,-178.440,9.981,149.561
C02455=1119.513,255.288,-71.591,-178.439,9.982,149.561
C02456=1119.509,255.537,-71.620,-178.439,9.984,149.562
C02457=1119.505,255.785,-71.649,-178.438,9.985,149.562
C02458=1119.500,256.033,-71.678,-178.437,9.987,149.562
C02459=1119.496,256.282,-71.706,-178.434,9.990,149.562
C02460=1119.492,256.530,-71.734,-178.431,9.993,149.562
C02461=1119.487,256.778,-71.764,-178.428,9.996,149.562
C02462=1119.483,257.026,-71.792,-178.425,9.998,149.562
C02463=1119.479,257.275,-71.821,-178.422,10.001,149.562
C02464=1119.475,257.524,-71.850,-178.420,10.004,149.561
C02465=1119.471,257.771,-71.878,-178.417,10.007,149.561
C02466=1119.466,258.020,-71.907,-178.414,10.010,149.561
C02467=1119.462,258.268,-71.937,-178.411,10.013,149.561
C02468=1119.457,258.516,-71.965,-178.408,10.015,149.561
C02469=1119.454,258.764,-71.994,-178.405,10.018,149.561
C02470=1119.449,259.013,-72.023,-178.402,10.021,149.561
C02471=1119.445,259.261,-72.052,-178.399,10.024,149.561
C02472=1119.441,259.510,-72.080,-178.396,10.026,149.561
C02473=1119.436,259.757,-72.109,-178.393,10.030,149.561
C02474=1119.432,260.006,-72.138,-178.390,10.033,149.561
C02475=1119.428,260.255,-72.167,-178.387,10.035,149.560
C02476=1119.424,260.503,-72.196,-178.384,10.038,149.560
C02477=1119.419,260.751,-72.225,-178.381,10.041,149.560
C02478=1119.415,260.999,-72.254,-178.377,10.044,149.560
C02479=1119.411,261.247,-72.284,-178.374,10.047,149.560
C02480=1119.406,261.496,-72.312,-178.371,10.050,149.560
C02481=1119.403,261.744,-72.341,-178.368,10.052,149.560
C02482=1119.399,261.992,-72.371,-178.365,10.056,149.560
C02483=1119.394,262.240,-72.400,-178.361,10.058,149.559
C02484=1119.389,262.489,-72.428,-178.358,10.061,149.559
C02485=1119.385,262.737,-72.458,-178.355,10.065,149.559
C02486=1119.381,262.985,-72.487,-178.351,10.067,149.559
C02487=1119.377,263.234,-72.517,-178.349,10.070,149.559
C02488=1119.372,263.483,-72.546,-178.345,10.073,149.559
C02489=1119.368,263.730,-72.574,-178.342,10.076,149.558
C02490=1119.364,263.978,-72.603,-178.339,10.078,149.558
C02491=1119.360,264.226,-72.633,-178.335,10.082,149.558
C02492=1119.356,264.475,-72.662,-178.331,10.084,149.558
C02493=1119.352,264.723,-72.692,-178.328,10.087,149.557
C02494=1119.347,264.971,-72.721,-178.326,10.089,149.557
C02495=1119.343,265.220,-72.750,-178.323,10.091,149.557
C02496=1119.339,265.468,-72.779,-178.321,10.094,149.557
C02497=1119.334,265.716,-72.809,-178.318,10.097,149.557
C02498=1119.330,265.964,-72.838,-178.315,10.099,149.557
C02499=1119.326,266.212,-72.867,-178.313,10.101,149.557
C02500=1119.322,266.426,-72.893,-178.311,10.103,149.557
C02501=1119.319,266.639,-72.919,-178.308,10.105,149.557
C02502=1119.315,266.852,-72.944,-178.306,10.107,149.557
C02503=1119.311,267.065,-72.969,-178.303,10.110,149.556
C02504=1119.307,267.278,-72.994,-178.301,10.112,149.556
C02505=1119.304,267.491,-73.020,-178.299,10.114,149.556
C02506=1119.301,267.704,-73.045,-178.297,10.116,149.556
C02507=1119.297,267.918,-73.070,-178.294,10.118,149.556
C02508=1119.292,268.165,-73.099,-178.291,10.121,149.556
C02509=1119.288,268.414,-73.129,-178.289,10.123,149.556
C02510=1119.284,268.662,-73.158,-178.286,10.126,149.556
C02511=1119.279,268.911,-73.188,-178.283,10.129,149.556
C02512=1119.275,269.158,-73.218,-178.280,10.131,149.556
C02513=1119.271,269.406,-73.248,-178.278,10.133,149.556
C02514=1119.267,269.655,-73.277,-178.275,10.136,149.555
C02515=1119.263,269.903,-73.307,-178.272,10.139,149.555
C02516=1119.258,270.151,-73.336,-178.269,10.142,149.555
C02517=1119.254,270.399,-73.365,-178.267,10.144,149.555
C02518=1119.250,270.647,-73.396,-178.264,10.146,149.555
C02519=1119.246,270.895,-73.425,-178.261,10.149,149.555
C02520=1119.241,271.144,-73.455,-178.258,10.152,149.555
C02521=1119.237,271.392,-73.485,-178.255,10.155,149.555
C02522=1119.233,271.641,-73.514,-178.253,10.157,149.555
C02523=1119.229,271.888,-73.544,-178.250,10.159,149.554
C02524=1119.225,272.136,-73.574,-178.247,10.162,149.554
C02525=1119.221,272.385,-73.603,-178.244,10.165,149.554
C02526=1119.217,272.633,-73.634,-178.241,10.168,149.554
C02527=1119.212,272.882,-73.664,-178.238,10.170,149.554
C02528=1119.208,273.130,-73.693,-178.235,10.173,149.554
C02529=1119.204,273.378,-73.723,-178.232,10.176,149.554
C02530=1119.199,273.626,-73.753,-178.229,10.178,149.554
C02531=1119.195,273.874,-73.783,-178.227,10.180,149.553
C02532=1119.191,274.122,-73.813,-178.224,10.183,149.553
C02533=1119.187,274.370,-73.842,-178.221,10.186,149.553
C02534=1119.182,274.619,-73.873,-178.217,10.188,149.553
C02535=1119.178,274.867,-73.903,-178.214,10.191,149.553
C02536=1119.174,275.115,-73.932,-178.212,10.194,149.553
C02537=1119.171,275.363,-73.963,-178.209,10.197,149.553
C02538=1119.166,275.612,-73.993,-178.206,10.199,149.553
C02539=1119.162,275.859,-74.023,-178.202,10.202,149.552
C02540=1119.158,276.108,-74.052,-178.199,10.204,149.552
C02541=1119.153,276.356,-74.083,-178.196,10.207,149.552
C02542=1119.149,276.604,-74.113,-178.194,10.210,149.552
C02543=1119.145,276.851,-74.143,-178.190,10.212,149.552
C02544=1119.141,277.101,-74.173,-178.187,10.215,149.552
C02545=1119.137,277.348,-74.203,-178.184,10.218,149.552
C02546=1119.133,277.597,-74.233,-178.181,10.221,149.551
C02547=1119.128,277.845,-74.264,-178.177,10.224,149.551
C02548=1119.124,278.092,-74.294,-178.174,10.227,149.551
C02549=1119.120,278.341,-74.324,-178.171,10.229,149.551
C02550=1119.116,278.589,-74.354,-178.168,10.232,149.551
C02551=1119.112,278.837,-74.384,-178.165,10.235,149.551
C02552=1119.107,279.085,-74.414,-178.162,10.237,149.550
C02553=1119.104,279.333,-74.445,-178.159,10.240,149.550
C02554=1119.099,279.581,-74.475,-178.156,10.242,149.550
C02555=1119.095,279.830,-74.505,-178.153,10.245,149.550
C02556=1119.091,280.043,-74.532,-178.150,10.248,149.550
C02557=1119.088,280.256,-74.558,-178.147,10.249,149.549
C02558=1119.085,280.469,-74.584,-178.144,10.252,149.549
C02559=1119.081,280.682,-74.610,-178.141,10.255,149.549
C02560=1119.078,280.895,-74.636,-178.138,10.256,149.549
C02561=1119.074,281.108,-74.662,-178.135,10.259,149.549
C02562=1119.070,281.321,-74.688,-178.133,10.261,149.549
C02563=1119.066,281.534,-74.715,-178.130,10.264,149.548
C02564=1119.062,281.782,-74.744,-178.127,10.266,149.548
C02565=1119.058,282.030,-74.775,-178.124,10.269,149.548
C02566=1119.054,282.278,-74.805,-178.121,10.272,149.548
C02567=1119.050,282.526,-74.836,-178.118,10.274,149.548
C02568=1119.046,282.774,-74.866,-178.115,10.276,149.548
C02569=1119.041,283.022,-74.897,-178.112,10.279,149.547
C02570=1119.037,283.270,-74.928,-178.109,10.281,149.547
C02571=1119.033,283.518,-74.959,-178.106,10.284,149.547
C02572=1119.028,283.767,-74.989,-178.103,10.287,149.547
C02573=1119.025,284.014,-75.019,-178.099,10.289,149.547
C02574=1119.021,284.263,-75.050,-178.097,10.292,149.547
C02575=1119.016,284.511,-75.081,-178.093,10.294,149.546
C02576=1119.012,284.759,-75.111,-178.091,10.296,149.546
C02577=1119.008,285.007,-75.142,-178.088,10.299,149.546
C02578=1119.003,285.255,-75.173,-178.085,10.301,149.546
C02579=1119.000,285.503,-75.203,-178.082,10.304,149.546
C02580=1118.996,285.752,-75.234,-178.078,10.307,149.546
C02581=1118.991,285.999,-75.265,-178.075,10.309,149.545
C02582=1118.987,286.246,-75.296,-178.072,10.312,149.545
C02583=1118.983,286.495,-75.327,-178.069,10.315,149.545
C02584=1118.979,286.743,-75.358,-178.066,10.317,149.545
C02585=1118.974,286.991,-75.388,-178.063,10.319,149.545
C02586=1118.971,287.239,-75.419,-178.061,10.322,149.545
C02587=1118.966,287.487,-75.450,-178.057,10.324,149.544
C02588=1118.962,287.735,-75.480,-178.054,10.327,149.544
C02589=1118.958,287.984,-75.511,-178.051,10.329,149.544
C02590=1118.954,288.231,-75.542,-178.048,10.332,149.544
C02591=1118.950,288.480,-75.574,-178.045,10.335,149.544
C02592=1118.945,288.728,-75.604,-178.042,10.337,149.543
C02593=1118.941,288.976,-75.635,-178.038,10.340,149.543
C02594=1118.938,289.224,-75.666,-178.036,10.342,149.543
C02595=1118.933,289.471,-75.697,-178.033,10.344,149.543
C02596=1118.929,289.720,-75.728,-178.030,10.347,149.543
C02597=1118.925,289.968,-75.759,-178.027,10.350,149.543
C02598=1118.921,290.216,-75.791,-178.024,10.352,149.542
C02599=1118.917,290.464,-75.821,-178.021,10.355,149.542
C02600=1118.913,290.712,-75.852,-178.017,10.357,149.542
C02601=1118.909,290.960,-75.884,-178.014,10.360,149.542
C02602=1118.904,291.208,-75.914,-178.011,10.362,149.542
C02603=1118.900,291.456,-75.945,-178.008,10.365,149.542
C02604=1118.896,291.704,-75.977,-178.005,10.367,149.541
C02605=1118.892,291.952,-76.008,-178.002,10.370,149.541
C02606=1118.887,292.200,-76.039,-177.999,10.372,149.541
C02607=1118.884,292.448,-76.070,-177.996,10.375,149.541
C02608=1118.880,292.696,-76.101,-177.993,10.378,149.541
C02609=1118.876,292.944,-76.133,-177.990,10.380,149.540
C02610=1118.871,293.192,-76.163,-177.987,10.383,149.540
C02611=1118.868,293.440,-76.195,-177.984,10.385,149.540
C02612=1118.864,293.653,-76.222,-177.981,10.387,149.540
C02613=1118.860,293.865,-76.249,-177.979,10.389,149.540
C02614=1118.856,294.079,-76.276,-177.976,10.392,149.540
C02615=1118.853,294.291,-76.302,-177.973,10.394,149.539
C02616=1118.850,294.504,-76.330,-177.971,10.396,149.539
C02617=1118.846,294.717,-76.356,-177.968,10.398,149.539
C02618=1118.843,294.930,-76.384,-177.965,10.400,149.539
C02619=1118.839,295.143,-76.410,-177.963,10.402,149.539
C02620=1118.834,295.391,-76.442,-177.960,10.405,149.539
C02621=1118.831,295.639,-76.474,-177.957,10.407,149.538
C02622=1118.827,295.887,-76.505,-177.954,10.410,149.538
C02623=1118.822,296.135,-76.536,-177.951,10.412,149.538
C02624=1118.819,296.383,-76.568,-177.948,10.415,149.538
C02625=1118.814,296.631,-76.599,-177.944,10.418,149.538
C02626=1118.810,296.879,-76.631,-177.941,10.420,149.538
C02627=1118.806,297.126,-76.662,-177.938,10.423,149.537
C02628=1118.802,297.375,-76.693,-177.935,10.426,149.537
C02629=1118.798,297.623,-76.725,-177.932,10.428,149.537
C02630=1118.794,297.870,-76.757,-177.929,10.430,149.537
C02631=1118.790,298.119,-76.788,-177.926,10.432,149.537
C02632=1118.786,298.366,-76.819,-177.923,10.435,149.537
C02633=1118.781,298.614,-76.852,-177.920,10.438,149.536
C02634=1118.778,298.862,-76.883,-177.917,10.440,149.536
C02635=1118.773,299.110,-76.914,-177.914,10.443,149.536
C02636=1118.769,299.358,-76.946,-177.911,10.446,149.536
C02637=1118.766,299.607,-76.978,-177.907,10.448,149.536
C02638=1118.761,299.854,-77.009,-177.904,10.451,149.536
C02639=1118.757,300.102,-77.042,-177.901,10.453,149.535
C02640=1118.753,300.350,-77.074,-177.899,10.455,149.535
C02641=1118.749,300.598,-77.105,-177.895,10.458,149.535
C02642=1118.745,300.846,-77.136,-177.893,10.460,149.535
C02643=1118.740,301.094,-77.168,-177.889,10.463,149.535
C02644=1118.736,301.342,-77.200,-177.886,10.466,149.535
C02645=1118.732,301.590,-77.232,-177.883,10.468,149.534
C02646=1118.728,301.837,-77.264,-177.880,10.471,149.534
C02647=1118.724,302.086,-77.296,-177.877,10.473,149.534
C02648=1118.720,302.334,-77.328,-177.874,10.476,149.534
C02649=1118.716,302.582,-77.360,-177.870,10.478,149.534
C02650=1118.712,302.829,-77.391,-177.867,10.481,149.533
C02651=1118.707,303.077,-77.424,-177.865,10.483,149.533
C02652=1118.704,303.325,-77.455,-177.862,10.486,149.533
C02653=1118.699,303.573,-77.487,-177.858,10.488,149.533
C02654=1118.695,303.821,-77.519,-177.856,10.491,149.533
C02655=1118.691,304.069,-77.551,-177.852,10.493,149.533
C02656=1118.688,304.317,-77.583,-177.849,10.496,149.532
C02657=1118.682,304.565,-77.615,-177.846,10.498,149.532
C02658=1118.679,304.812,-77.648,-177.843,10.501,149.532
C02659=1118.675,305.060,-77.680,-177.840,10.504,149.532
C02660=1118.671,305.309,-77.712,-177.836,10.506,149.532
C02661=1118.667,305.556,-77.743,-177.833,10.509,149.531
C02662=1118.662,305.804,-77.776,-177.831,10.510,149.531
C02663=1118.658,306.052,-77.808,-177.828,10.513,149.531
C02664=1118.655,306.300,-77.840,-177.824,10.516,149.531
C02665=1118.650,306.547,-77.872,-177.822,10.518,149.531
C02666=1118.646,306.796,-77.904,-177.818,10.521,149.531
C02667=1118.642,307.044,-77.937,-177.815,10.524,149.530
C02668=1118.638,307.256,-77.964,-177.813,10.525,149.530
C02669=1118.635,307.469,-77.992,-177.810,10.528,149.530
C02670=1118.632,307.681,-78.019,-177.807,10.530,149.530
C02671=1118.628,307.895,-78.048,-177.805,10.532,149.530
C02672=1118.624,308.107,-78.075,-177.802,10.535,149.530
C02673=1118.621,308.320,-78.103,-177.799,10.537,149.530
C02674=1118.618,308.532,-78.130,-177.797,10.538,149.529
C02675=1118.615,308.746,-78.158,-177.794,10.541,149.529
C02676=1118.610,308.993,-78.191,-177.790,10.543,149.529
C02677=1118.606,309.241,-78.222,-177.788,10.546,149.529
C02678=1118.602,309.489,-78.255,-177.784,10.549,149.529
C02679=1118.598,309.736,-78.287,-177.782,10.551,149.528
C02680=1118.594,309.985,-78.320,-177.779,10.553,149.528
C02681=1118.590,310.233,-78.353,-177.776,10.556,149.528
C02682=1118.586,310.481,-78.385,-177.772,10.558,149.528
C02683=1118.581,310.728,-78.418,-177.769,10.561,149.528
C02684=1118.578,310.976,-78.450,-177.766,10.563,149.528
C02685=1118.573,311.223,-78.483,-177.763,10.566,149.527
C02686=1118.570,311.471,-78.515,-177.760,10.569,149.527
C02687=1118.566,311.719,-78.548,-177.756,10.571,149.527
C02688=1118.561,311.967,-78.580,-177.754,10.574,149.527
C02689=1118.558,312.215,-78.613,-177.750,10.576,149.527
C02690=1118.553,312.463,-78.645,-177.747,10.579,149.527
C02691=1118.550,312.711,-78.678,-177.745,10.581,149.526
C02692=1118.545,312.959,-78.710,-177.741,10.583,149.526
C02693=1118.541,313.207,-78.743,-177.738,10.586,149.526
C02694=1118.538,313.455,-78.775,-177.735,10.588,149.526
C02695=1118.533,313.702,-78.808,-177.732,10.591,149.526
C02696=1118.529,313.950,-78.841,-177.729,10.594,149.525
C02697=1118.525,314.198,-78.873,-177.725,10.596,149.525
C02698=1118.521,314.445,-78.906,-177.723,10.599,149.525
C02699=1118.517,314.693,-78.939,-177.719,10.601,149.525
C02700=1118.512,314.941,-78.972,-177.716,10.604,149.525
C02701=1118.509,315.189,-79.004,-177.713,10.606,149.524
C02702=1118.505,315.437,-79.037,-177.710,10.609,149.524
C02703=1118.501,315.684,-79.071,-177.707,10.611,149.524
C02704=1118.497,315.932,-79.102,-177.704,10.613,149.524
C02705=1118.493,316.180,-79.136,-177.701,10.616,149.524
C02706=1118.489,316.428,-79.169,-177.698,10.619,149.524
C02707=1118.485,316.675,-79.202,-177.694,10.621,149.523
C02708=1118.481,316.923,-79.234,-177.691,10.624,149.523
C02709=1118.477,317.171,-79.267,-177.688,10.626,149.523
C02710=1118.473,317.419,-79.300,-177.685,10.629,149.523
C02711=1118.468,317.667,-79.333,-177.682,10.631,149.523
C02712=1118.465,317.915,-79.367,-177.679,10.634,149.522
C02713=1118.461,318.163,-79.399,-177.676,10.637,149.522
C02714=1118.457,318.410,-79.432,-177.672,10.639,149.522
C02715=1118.453,318.658,-79.466,-177.670,10.641,149.522
C02716=1118.449,318.906,-79.498,-177.667,10.643,149.522
C02717=1118.445,319.154,-79.531,-177.663,10.646,149.521
C02718=1118.440,319.402,-79.564,-177.660,10.649,149.521
C02719=1118.437,319.649,-79.597,-177.657,10.651,149.521
C02720=1118.433,319.897,-79.630,-177.654,10.654,149.521
C02721=1118.429,320.145,-79.663,-177.651,10.656,149.521
C02722=1118.425,320.392,-79.696,-177.648,10.659,149.521
C02723=1118.421,320.640,-79.729,-177.645,10.662,149.520
C02724=1118.417,320.853,-79.758,-177.642,10.663,149.520
C02725=1118.414,321.066,-79.787,-177.639,10.666,149.520
C02726=1118.410,321.278,-79.815,-177.636,10.668,149.520
C02727=1118.407,321.490,-79.843,-177.634,10.670,149.520
C02728=1118.404,321.703,-79.872,-177.631,10.672,149.520
C02729=1118.400,321.915,-79.900,-177.628,10.674,149.519
C02730=1118.397,322.128,-79.929,-177.626,10.676,149.519
C02731=1118.393,322.341,-79.958,-177.623,10.679,149.519
C02732=1118.389,322.589,-79.991,-177.620,10.681,149.519
C02733=1118.385,322.836,-80.024,-177.617,10.684,149.519
C02734=1118.381,323.083,-80.058,-177.614,10.685,149.518
C02735=1118.377,323.331,-80.091,-177.611,10.688,149.518
C02736=1118.374,323.580,-80.125,-177.608,10.691,149.518
C02737=1118.369,323.827,-80.158,-177.604,10.693,149.518
C02738=1118.365,324.075,-80.191,-177.601,10.696,149.518
C02739=1118.361,324.322,-80.225,-177.598,10.698,149.518
C02740=1118.357,324.570,-80.258,-177.595,10.701,149.517
C02741=1118.354,324.818,-80.292,-177.592,10.704,149.517
C02742=1118.350,325.066,-80.325,-177.588,10.706,149.517
C02743=1118.346,325.313,-80.359,-177.585,10.708,149.517
C02744=1118.342,325.561,-80.392,-177.582,10.711,149.517
C02745=1118.338,325.809,-80.425,-177.579,10.714,149.517
C02746=1118.334,326.056,-80.459,-177.576,10.715,149.516
C02747=1118.330,326.304,-80.493,-177.573,10.718,149.516
C02748=1118.326,326.552,-80.526,-177.570,10.721,149.516
C02749=1118.322,326.799,-80.560,-177.567,10.723,149.516
C02750=1118.318,327.048,-80.594,-177.564,10.726,149.516
C02751=1118.314,327.295,-80.627,-177.560,10.728,149.515
C02752=1118.310,327.543,-80.661,-177.557,10.731,149.515
C02753=1118.306,327.790,-80.694,-177.554,10.734,149.515
C02754=1118.302,328.037,-80.728,-177.551,10.736,149.515
C02755=1118.298,328.286,-80.761,-177.548,10.738,149.515
C02756=1118.294,328.533,-80.796,-177.545,10.741,149.515
C02757=1118.290,328.781,-80.829,-177.541,10.744,149.514
C02758=1118.287,329.029,-80.863,-177.538,10.746,149.514
C02759=1118.282,329.277,-80.896,-177.536,10.748,149.514
C02760=1118.278,329.524,-80.931,-177.532,10.751,149.514
C02761=1118.274,329.772,-80.964,-177.529,10.753,149.513
C02762=1118.270,330.019,-80.998,-177.526,10.755,149.513
C02763=1118.266,330.267,-81.031,-177.523,10.758,149.513
C02764=1118.262,330.515,-81.066,-177.519,10.761,149.513
C02765=1118.258,330.763,-81.099,-177.516,10.763,149.513
C02766=1118.254,331.010,-81.133,-177.513,10.766,149.513
C02767=1118.251,331.257,-81.167,-177.510,10.768,149.512
C02768=1118.246,331.506,-81.201,-177.507,10.771,149.512
C02769=1118.242,331.753,-81.235,-177.504,10.774,149.512
C02770=1118.239,332.000,-81.269,-177.500,10.776,149.512
C02771=1118.234,332.249,-81.303,-177.497,10.778,149.512
C02772=1118.231,332.496,-81.337,-177.494,10.780,149.511
C02773=1118.227,332.743,-81.371,-177.491,10.783,149.511
C02774=1118.222,332.992,-81.405,-177.488,10.785,149.511
C02775=1118.219,333.239,-81.439,-177.485,10.788,149.511
C02776=1118.215,333.487,-81.473,-177.481,10.790,149.511
C02777=1118.211,333.734,-81.507,-177.479,10.793,149.511
C02778=1118.207,333.981,-81.541,-177.475,10.796,149.510
C02779=1118.203,334.230,-81.575,-177.472,10.798,149.510
C02780=1118.200,334.442,-81.604,-177.470,10.800,149.510
C02781=1118.196,334.654,-81.634,-177.466,10.802,149.510
C02782=1118.193,334.866,-81.663,-177.464,10.804,149.510
C02783=1118.190,335.079,-81.692,-177.461,10.806,149.509
C02784=1118.186,335.291,-81.722,-177.458,10.809,149.509
C02785=1118.183,335.504,-81.751,-177.456,10.811,149.509
C02786=1118.180,335.716,-81.780,-177.453,10.813,149.509
C02787=1118.176,335.928,-81.810,-177.450,10.815,149.509
C02788=1118.172,336.176,-81.844,-177.447,10.818,149.509
C02789=1118.168,336.424,-81.878,-177.444,10.820,149.508
C02790=1118.164,336.672,-81.912,-177.441,10.823,149.508
C02791=1118.161,336.919,-81.946,-177.437,10.825,149.508
C02792=1118.156,337.167,-81.981,-177.435,10.827,149.508
C02793=1118.153,337.415,-82.015,-177.432,10.830,149.508
C02794=1118.148,337.662,-82.050,-177.428,10.832,149.507
C02795=1118.145,337.910,-82.084,-177.425,10.835,149.507
C02796=1118.140,338.157,-82.118,-177.422,10.837,149.507
C02797=1118.137,338.404,-82.152,-177.419,10.840,149.507
C02798=1118.133,338.653,-82.187,-177.415,10.842,149.507
C02799=1118.128,338.900,-82.222,-177.412,10.845,149.506
C02800=1118.125,339.148,-82.256,-177.409,10.847,149.506
C02801=1118.121,339.395,-82.291,-177.406,10.850,149.506
C02802=1118.117,339.642,-82.325,-177.403,10.852,149.506
C02803=1118.113,339.890,-82.360,-177.399,10.855,149.506
C02804=1118.109,340.138,-82.394,-177.396,10.857,149.505
C02805=1118.105,340.385,-82.428,-177.394,10.859,149.505
C02806=1118.101,340.633,-82.463,-177.390,10.862,149.505
C02807=1118.096,340.881,-82.498,-177.387,10.864,149.505
C02808=1118.093,341.128,-82.533,-177.384,10.867,149.505
C02809=1118.089,341.375,-82.567,-177.380,10.869,149.504
C02810=1118.085,341.623,-82.602,-177.377,10.872,149.504
C02811=1118.082,341.871,-82.636,-177.374,10.874,149.504
C02812=1118.077,342.118,-82.671,-177.371,10.877,149.504
C02813=1118.073,342.366,-82.706,-177.368,10.879,149.504
C02814=1118.070,342.613,-82.740,-177.364,10.882,149.503
C02815=1118.066,342.861,-82.775,-177.361,10.885,149.503
C02816=1118.061,343.108,-82.810,-177.358,10.887,149.503
C02817=1118.058,343.356,-82.844,-177.355,10.889,149.503
C02818=1118.054,343.604,-82.879,-177.352,10.891,149.503
C02819=1118.050,343.851,-82.914,-177.349,10.894,149.502
C02820=1118.046,344.099,-82.949,-177.346,10.896,149.502
C02821=1118.041,344.346,-82.984,-177.342,10.899,149.502
C02822=1118.038,344.594,-83.019,-177.339,10.901,149.502
C02823=1118.035,344.842,-83.053,-177.336,10.904,149.502
C02824=1118.030,345.088,-83.089,-177.332,10.906,149.501
C02825=1118.026,345.337,-83.123,-177.329,10.909,149.501
C02826=1118.023,345.583,-83.158,-177.326,10.911,149.501
C02827=1118.019,345.831,-83.193,-177.323,10.914,149.501
C02828=1118.015,346.079,-83.228,-177.320,10.916,149.501
C02829=1118.011,346.326,-83.263,-177.316,10.919,149.500
C02830=1118.007,346.574,-83.298,-177.313,10.921,149.500
C02831=1118.003,346.822,-83.333,-177.310,10.924,149.500
C02832=1117.999,347.068,-83.368,-177.307,10.926,149.500
C02833=1117.995,347.316,-83.403,-177.304,10.928,149.500
C02834=1117.992,347.564,-83.438,-177.301,10.931,149.499
C02835=1117.987,347.811,-83.473,-177.297,10.933,149.499
C02836=1117.984,348.023,-83.503,-177.294,10.936,149.499
C02837=1117.981,348.236,-83.534,-177.292,10.938,149.499
C02838=1117.978,348.448,-83.563,-177.289,10.939,149.499
C02839=1117.974,348.660,-83.594,-177.286,10.942,149.499
C02840=1117.971,348.873,-83.624,-177.284,10.944,149.498
C02841=1117.968,349.085,-83.653,-177.281,10.945,149.498
C02842=1117.964,349.297,-83.684,-177.278,10.948,149.498
C02843=1117.961,349.509,-83.714,-177.275,10.950,149.498
C02844=1117.957,349.757,-83.749,-177.272,10.952,149.498
C02845=1117.953,350.005,-83.784,-177.269,10.955,149.497
C02846=1117.949,350.252,-83.820,-177.265,10.958,149.497
C02847=1117.945,350.499,-83.855,-177.261,10.961,149.497
C02848=1117.942,350.746,-83.890,-177.258,10.963,149.497
C02849=1117.938,350.995,-83.925,-177.255,10.965,149.496
C02850=1117.934,351.242,-83.961,-177.252,10.968,149.496
C02851=1117.930,351.489,-83.996,-177.248,10.970,149.496
C02852=1117.926,351.736,-84.031,-177.244,10.974,149.496
C02853=1117.922,351.984,-84.067,-177.241,10.976,149.495
C02854=1117.919,352.231,-84.103,-177.237,10.978,149.495
C02855=1117.914,352.479,-84.137,-177.234,10.981,149.495
C02856=1117.910,352.726,-84.173,-177.231,10.983,149.495
C02857=1117.907,352.974,-84.208,-177.227,10.986,149.495
C02858=1117.903,353.221,-84.244,-177.224,10.988,149.494
C02859=1117.899,353.469,-84.280,-177.221,10.991,149.494
C02860=1117.895,353.717,-84.315,-177.217,10.993,149.494
C02861=1117.891,353.963,-84.351,-177.213,10.996,149.494
C02862=1117.887,354.211,-84.386,-177.210,10.998,149.493
C02863=1117.883,354.458,-84.422,-177.206,11.001,149.493
C02864=1117.880,354.706,-84.457,-177.203,11.003,149.493
C02865=1117.876,354.953,-84.493,-177.200,11.006,149.493
C02866=1117.872,355.201,-84.528,-177.197,11.008,149.492
C02867=1117.868,355.448,-84.563,-177.193,11.010,149.492
C02868=1117.864,355.696,-84.600,-177.190,11.013,149.492
C02869=1117.860,355.943,-84.635,-177.186,11.015,149.492
C02870=1117.856,356.191,-84.671,-177.183,11.018,149.491
C02871=1117.853,356.438,-84.706,-177.180,11.020,149.491
C02872=1117.849,356.685,-84.743,-177.176,11.022,149.491
C02873=1117.846,356.932,-84.778,-177.173,11.025,149.490
C02874=1117.841,357.180,-84.814,-177.169,11.027,149.490
C02875=1117.838,357.428,-84.850,-177.166,11.030,149.490
C02876=1117.834,357.675,-84.885,-177.163,11.032,149.490
C02877=1117.830,357.922,-84.921,-177.159,11.034,149.489
C02878=1117.826,358.169,-84.957,-177.156,11.037,149.489
C02879=1117.822,358.417,-84.993,-177.152,11.040,149.489
C02880=1117.818,358.664,-85.028,-177.148,11.043,149.489
C02881=1117.815,358.912,-85.064,-177.145,11.045,149.488
C02882=1117.811,359.159,-85.101,-177.141,11.047,149.488
C02883=1117.807,359.406,-85.136,-177.138,11.050,149.488
C02884=1117.803,359.654,-85.172,-177.135,11.052,149.488
C02885=1117.799,359.901,-85.209,-177.131,11.055,149.488
C02886=1117.796,360.149,-85.244,-177.128,11.057,149.487
C02887=1117.792,360.396,-85.280,-177.124,11.059,149.487
C02888=1117.789,360.643,-85.316,-177.121,11.062,149.487
C02889=1117.784,360.891,-85.352,-177.118,11.064,149.486
C02890=1117.780,361.138,-85.388,-177.115,11.067,149.486
C02891=1117.776,361.386,-85.425,-177.111,11.069,149.486
C02892=1117.773,361.597,-85.455,-177.108,11.070,149.486
C02893=1117.770,361.810,-85.486,-177.106,11.072,149.486
C02894=1117.767,362.022,-85.517,-177.103,11.075,149.485
C02895=1117.764,362.234,-85.549,-177.100,11.077,149.485
C02896=1117.761,362.446,-85.579,-177.097,11.079,149.485
C02897=1117.757,362.658,-85.610,-177.094,11.081,149.485
C02898=1117.754,362.871,-85.641,-177.091,11.082,149.484
C02899=1117.751,363.083,-85.672,-177.088,11.085,149.484
C02900=1117.747,363.329,-85.708,-177.085,11.087,149.484
C02901=1117.743,363.577,-85.745,-177.081,11.090,149.484
C02902=1117.739,363.824,-85.781,-177.078,11.092,149.483
C02903=1117.735,364.071,-85.817,-177.074,11.094,149.483
C02904=1117.732,364.319,-85.853,-177.071,11.097,149.483
C02905=1117.728,364.566,-85.889,-177.068,11.099,149.483
C02906=1117.724,364.814,-85.926,-177.064,11.102,149.482
C02907=1117.721,365.061,-85.962,-177.062,11.104,149.482
C02908=1117.717,365.308,-85.999,-177.058,11.106,149.482
C02909=1117.713,365.556,-86.035,-177.055,11.108,149.482
C02910=1117.709,365.803,-86.071,-177.051,11.111,149.481
C02911=1117.705,366.050,-86.108,-177.048,11.113,149.481
C02912=1117.702,366.298,-86.144,-177.045,11.116,149.481
C02913=1117.697,366.545,-86.181,-177.041,11.118,149.481
C02914=1117.694,366.792,-86.217,-177.038,11.120,149.480
C02915=1117.690,367.039,-86.254,-177.035,11.123,149.480
C02916=1117.687,367.287,-86.290,-177.031,11.125,149.480
C02917=1117.683,367.534,-86.326,-177.028,11.128,149.480
C02918=1117.679,367.781,-86.363,-177.025,11.130,149.480
C02919=1117.675,368.028,-86.400,-177.021,11.133,149.479
C02920=1117.671,368.276,-86.436,-177.018,11.135,149.479
C02921=1117.668,368.523,-86.472,-177.014,11.137,149.479
C02922=1117.664,368.770,-86.509,-177.011,11.140,149.478
C02923=1117.660,369.018,-86.546,-177.008,11.141,149.478
C02924=1117.657,369.265,-86.582,-177.005,11.144,149.478
C02925=1117.653,369.512,-86.619,-177.002,11.146,149.478
C02926=1117.648,369.759,-86.656,-176.998,11.149,149.478
C02927=1117.645,370.006,-86.692,-176.995,11.151,149.477
C02928=1117.641,370.253,-86.729,-176.992,11.154,149.477
C02929=1117.638,370.501,-86.766,-176.989,11.156,149.477
C02930=1117.634,370.748,-86.803,-176.985,11.159,149.477
C02931=1117.630,370.995,-86.840,-176.982,11.161,149.476
C02932=1117.626,371.243,-86.876,-176.978,11.163,149.476
C02933=1117.622,371.490,-86.913,-176.975,11.166,149.476
C02934=1117.619,371.737,-86.950,-176.972,11.168,149.476
C02935=1117.615,371.985,-86.987,-176.969,11.170,149.476
C02936=1117.611,372.232,-87.024,-176.966,11.172,149.475
C02937=1117.607,372.479,-87.060,-176.962,11.175,149.475
C02938=1117.604,372.727,-87.097,-176.959,11.177,149.475
C02939=1117.600,372.974,-87.134,-176.956,11.180,149.475
C02940=1117.596,373.221,-87.171,-176.953,11.182,149.475
C02941=1117.592,373.468,-87.208,-176.949,11.185,149.474
C02942=1117.589,373.716,-87.244,-176.946,11.187,149.474
C02943=1117.585,373.962,-87.282,-176.943,11.190,149.474
C02944=1117.581,374.209,-87.319,-176.940,11.193,149.474
C02945=1117.578,374.457,-87.356,-176.936,11.195,149.474
C02946=1117.574,374.705,-87.393,-176.933,11.198,149.473
C02947=1117.569,374.952,-87.430,-176.930,11.199,149.473
C02948=1117.567,375.164,-87.462,-176.927,11.202,149.473
C02949=1117.563,375.375,-87.493,-176.925,11.204,149.473
C02950=1117.561,375.587,-87.525,-176.922,11.206,149.473
C02951=1117.557,375.799,-87.556,-176.919,11.208,149.473
C02952=1117.554,376.011,-87.589,-176.917,11.210,149.472
C02953=1117.551,376.223,-87.621,-176.913,11.213,149.472
C02954=1117.547,376.435,-87.652,-176.911,11.215,149.472
C02955=1117.545,376.647,-87.684,-176.908,11.216,149.472
C02956=1117.541,376.894,-87.721,-176.905,11.219,149.472
C02957=1117.537,377.142,-87.758,-176.902,11.221,149.472
C02958=1117.533,377.388,-87.796,-176.899,11.224,149.472
C02959=1117.529,377.636,-87.833,-176.896,11.226,149.471
C02960=1117.526,377.884,-87.870,-176.892,11.229,149.471
C02961=1117.522,378.130,-87.908,-176.889,11.231,149.471
C02962=1117.518,378.377,-87.945,-176.886,11.234,149.471
C02963=1117.515,378.625,-87.982,-176.883,11.237,149.471
C02964=1117.511,378.872,-88.019,-176.880,11.239,149.471
C02965=1117.507,379.118,-88.057,-176.876,11.242,149.470
C02966=1117.503,379.366,-88.094,-176.874,11.244,149.470
C02967=1117.500,379.613,-88.132,-176.871,11.246,149.470
C02968=1117.496,379.861,-88.169,-176.867,11.249,149.470
C02969=1117.492,380.107,-88.206,-176.865,11.252,149.470
C02970=1117.488,380.354,-88.243,-176.861,11.254,149.470
C02971=1117.485,380.602,-88.281,-176.858,11.257,149.470
C02972=1117.481,380.849,-88.318,-176.855,11.259,149.469
C02973=1117.478,381.096,-88.356,-176.852,11.262,149.469
C02974=1117.474,381.343,-88.393,-176.849,11.265,149.469
C02975=1117.470,381.590,-88.431,-176.846,11.267,149.469
C02976=1117.467,381.837,-88.468,-176.843,11.270,149.469
C02977=1117.462,382.085,-88.506,-176.839,11.272,149.469
C02978=1117.459,382.332,-88.544,-176.836,11.275,149.469
C02979=1117.455,382.579,-88.581,-176.833,11.278,149.469
C02980=1117.451,382.826,-88.619,-176.830,11.281,149.469
C02981=1117.448,383.073,-88.656,-176.828,11.282,149.468
C02982=1117.444,383.320,-88.694,-176.825,11.285,149.468
C02983=1117.440,383.567,-88.731,-176.822,11.288,149.468
C02984=1117.437,383.815,-88.769,-176.820,11.290,149.468
C02985=1117.433,384.062,-88.807,-176.817,11.292,149.468
C02986=1117.429,384.309,-88.844,-176.815,11.294,149.468
C02987=1117.425,384.556,-88.882,-176.813,11.297,149.468
C02988=1117.422,384.803,-88.920,-176.810,11.299,149.468
C02989=1117.418,385.050,-88.957,-176.808,11.301,149.468
C02990=1117.415,385.297,-88.995,-176.806,11.304,149.468
C02991=1117.410,385.545,-89.033,-176.803,11.306,149.468
C02992=1117.407,385.792,-89.071,-176.801,11.309,149.469
C02993=1117.403,386.038,-89.108,-176.799,11.311,149.469
C02994=1117.400,386.286,-89.146,-176.797,11.313,149.469
C02995=1117.396,386.532,-89.184,-176.794,11.316,149.469
C02996=1117.392,386.780,-89.222,-176.792,11.318,149.469
C02997=1117.389,387.026,-89.260,-176.791,11.321,149.469
C02998=1117.385,387.274,-89.297,-176.788,11.323,149.469
C02999=1117.381,387.521,-89.335,-176.786,11.326,149.469
C03000=1117.377,387.769,-89.373,-176.784,11.328,149.469
C03001=1117.374,388.015,-89.411,-176.781,11.331,149.469
C03002=1117.370,388.262,-89.449,-176.780,11.334,149.470
C03003=1117.367,388.510,-89.487,-176.778,11.336,149.470
C03004=1117.363,388.721,-89.519,-176.775,11.338,149.470
C03005=1117.361,388.933,-89.552,-176.774,11.340,149.470
C03006=1117.357,389.145,-89.584,-176.772,11.343,149.470
C03007=1117.354,389.357,-89.618,-176.770,11.345,149.470
C03008=1117.351,389.569,-89.650,-176.768,11.348,149.470
C03009=1117.347,389.780,-89.682,-176.766,11.350,149.470
C03010=1117.345,389.992,-89.714,-176.765,11.353,149.471
C03011=1117.341,390.204,-89.747,-176.763,11.355,149.471
C03012=1117.338,390.451,-89.785,-176.761,11.357,149.471
C03013=1117.334,390.698,-89.823,-176.758,11.360,149.471
C03014=1117.331,390.945,-89.862,-176.757,11.363,149.471
C03015=1117.327,391.191,-89.899,-176.754,11.366,149.472
C03016=1117.324,391.439,-89.937,-176.753,11.369,149.472
C03017=1117.320,391.686,-89.976,-176.750,11.372,149.472
C03018=1117.316,391.933,-90.013,-176.748,11.374,149.472
C03019=1117.313,392.180,-90.051,-176.746,11.378,149.473
C03020=1117.309,392.428,-90.090,-176.745,11.381,149.473
C03021=1117.305,392.674,-90.127,-176.742,11.384,149.473
C03022=1117.301,392.922,-90.166,-176.741,11.386,149.473
C03023=1117.298,393.168,-90.204,-176.739,11.390,149.474
C03024=1117.295,393.415,-90.242,-176.736,11.393,149.474
C03025=1117.291,393.663,-90.281,-176.735,11.396,149.474
C03026=1117.287,393.909,-90.318,-176.733,11.399,149.475
C03027=1117.283,394.157,-90.357,-176.731,11.402,149.475
C03028=1117.280,394.404,-90.396,-176.729,11.405,149.475
C03029=1117.276,394.650,-90.434,-176.727,11.409,149.476
C03030=1117.272,394.898,-90.472,-176.725,11.412,149.476
C03031=1117.268,395.145,-90.510,-176.723,11.415,149.476
C03032=1117.265,395.391,-90.548,-176.721,11.418,149.477
C03033=1117.261,395.639,-90.587,-176.719,11.422,149.477
C03034=1117.258,395.886,-90.625,-176.718,11.425,149.477
C03035=1117.253,396.133,-90.663,-176.716,11.428,149.478
C03036=1117.250,396.380,-90.702,-176.714,11.432,149.478
C03037=1117.246,396.627,-90.740,-176.712,11.435,149.479
C03038=1117.243,396.874,-90.778,-176.711,11.438,149.479
C03039=1117.239,397.121,-90.817,-176.709,11.442,149.480
C03040=1117.236,397.368,-90.855,-176.707,11.446,149.480
C03041=1117.232,397.615,-90.894,-176.705,11.449,149.481
C03042=1117.228,397.862,-90.932,-176.703,11.453,149.481
C03043=1117.225,398.109,-90.970,-176.701,11.457,149.482
C03044=1117.222,398.356,-91.009,-176.699,11.460,149.482
C03045=1117.218,398.603,-91.048,-176.698,11.463,149.483
C03046=1117.214,398.849,-91.086,-176.696,11.467,149.483
C03047=1117.210,399.097,-91.124,-176.695,11.471,149.484
C03048=1117.207,399.344,-91.163,-176.693,11.475,149.484
C03049=1117.204,399.591,-91.202,-176.691,11.478,149.485
C03050=1117.199,399.837,-91.241,-176.690,11.482,149.485
C03051=1117.196,400.085,-91.278,-176.688,11.486,149.486
C03052=1117.193,400.332,-91.318,-176.686,11.490,149.486
C03053=1117.189,400.579,-91.356,-176.684,11.494,149.487
C03054=1117.185,400.825,-91.395,-176.683,11.497,149.488
C03055=1117.181,401.073,-91.433,-176.681,11.501,149.488
C03056=1117.178,401.319,-91.472,-176.680,11.505,149.489
C03057=1117.174,401.567,-91.510,-176.678,11.509,149.490
C03058=1117.171,401.814,-91.550,-176.677,11.513,149.490
C03059=1117.167,402.060,-91.587,-176.675,11.517,149.491
C03060=1117.164,402.272,-91.620,-176.673,11.521,149.491
C03061=1117.161,402.484,-91.654,-176.672,11.525,149.492
C03062=1117.157,402.696,-91.687,-176.671,11.528,149.492
C03063=1117.154,402.907,-91.720,-176.669,11.532,149.493
C03064=1117.152,403.119,-91.753,-176.668,11.535,149.494
C03065=1117.149,403.330,-91.786,-176.667,11.539,149.494
C03066=1117.146,403.542,-91.820,-176.666,11.542,149.495
C03067=1117.142,403.754,-91.853,-176.664,11.546,149.496
C03068=1117.139,404.001,-91.892,-176.663,11.550,149.496
C03069=1117.136,404.247,-91.931,-176.661,11.555,149.497
C03070=1117.132,404.494,-91.970,-176.659,11.559,149.498
C03071=1117.128,404.742,-92.009,-176.659,11.564,149.499
C03072=1117.124,404.988,-92.047,-176.657,11.568,149.499
C03073=1117.121,405.235,-92.086,-176.655,11.573,149.500
C03074=1117.118,405.482,-92.125,-176.654,11.577,149.501
C03075=1117.114,405.729,-92.164,-176.653,11.581,149.502
C03076=1117.110,405.976,-92.203,-176.651,11.586,149.503
C03077=1117.107,406.223,-92.242,-176.650,11.591,149.504
C03078=1117.104,406.470,-92.281,-176.649,11.595,149.504
C03079=1117.100,406.717,-92.320,-176.647,11.600,149.505
C03080=1117.095,406.964,-92.359,-176.646,11.604,149.506
C03081=1117.093,407.211,-92.397,-176.644,11.609,149.507
C03082=1117.089,407.457,-92.436,-176.643,11.614,149.508
C03083=1117.085,407.704,-92.476,-176.642,11.619,149.509
C03084=1117.082,407.951,-92.515,-176.641,11.623,149.510
C03085=1117.078,408.198,-92.554,-176.639,11.629,149.511
C03086=1117.074,408.445,-92.593,-176.638,11.633,149.512
C03087=1117.072,408.692,-92.632,-176.637,11.638,149.513
C03088=1117.068,408.939,-92.671,-176.636,11.643,149.514
C03089=1117.064,409.186,-92.711,-176.635,11.648,149.515
C03090=1117.061,409.433,-92.750,-176.634,11.653,149.516
C03091=1117.057,409.680,-92.789,-176.632,11.658,149.517
C03092=1117.053,409.927,-92.828,-176.631,11.663,149.518
C03093=1117.050,410.174,-92.868,-176.630,11.668,149.519
C03094=1117.046,410.420,-92.906,-176.629,11.673,149.520
C03095=1117.043,410.667,-92.945,-176.627,11.679,149.521
C03096=1117.039,410.914,-92.984,-176.627,11.683,149.522
C03097=1117.036,411.161,-93.024,-176.625,11.689,149.523
C03098=1117.032,411.408,-93.063,-176.624,11.695,149.524
C03099=1117.028,411.654,-93.102,-176.623,11.700,149.525
C03100=1117.025,411.901,-93.141,-176.622,11.705,149.527
C03101=1117.021,412.148,-93.181,-176.621,11.710,149.528
C03102=1117.017,412.395,-93.220,-176.620,11.716,149.529
C03103=1117.014,412.642,-93.259,-176.619,11.721,149.530
C03104=1117.010,412.889,-93.299,-176.618,11.727,149.531
C03105=1117.007,413.136,-93.338,-176.617,11.733,149.533
C03106=1117.003,413.383,-93.378,-176.616,11.738,149.534
C03107=1117.000,413.630,-93.417,-176.615,11.744,149.535
C03108=1116.997,413.877,-93.456,-176.614,11.749,149.536
C03109=1116.995,414.123,-93.495,-176.613,11.755,149.537
C03110=1116.992,414.370,-93.534,-176.612,11.761,149.539
C03111=1116.991,414.617,-93.574,-176.611,11.766,149.540
C03112=1116.991,414.864,-93.613,-176.610,11.772,149.541
C03113=1116.990,415.111,-93.652,-176.610,11.778,149.543
C03114=1116.990,415.358,-93.691,-176.609,11.784,149.544
C03115=1116.990,415.605,-93.730,-176.608,11.790,149.545
C03116=1116.992,415.817,-93.763,-176.608,11.795,149.547
C03117=1116.993,416.027,-93.797,-176.607,11.800,149.548
C03118=1116.995,416.239,-93.829,-176.606,11.805,149.549
C03119=1116.997,416.451,-93.863,-176.606,11.810,149.550
C03120=1117.000,416.662,-93.896,-176.605,11.815,149.551
C03121=1117.002,416.873,-93.929,-176.604,11.821,149.553
C03122=1117.006,417.085,-93.962,-176.604,11.826,149.554
C03123=1117.010,417.296,-93.995,-176.604,11.831,149.555
C03124=1116.590,417.296,-94.057,-176.596,11.836,149.554
C03125=1116.588,417.085,-94.025,-176.597,11.830,149.553
C03126=1116.584,416.873,-93.991,-176.597,11.825,149.552
C03127=1116.581,416.662,-93.958,-176.598,11.821,149.551
C03128=1116.577,416.450,-93.925,-176.598,11.815,149.549
C03129=1116.576,416.239,-93.892,-176.599,11.810,149.548
C03130=1116.574,416.027,-93.859,-176.600,11.804,149.547
C03131=1116.573,415.816,-93.825,-176.600,11.799,149.546
C03132=1116.572,415.604,-93.792,-176.601,11.794,149.545
C03133=1116.571,415.358,-93.753,-176.602,11.789,149.543
C03134=1116.571,415.112,-93.714,-176.603,11.783,149.542
C03135=1116.572,414.864,-93.676,-176.603,11.777,149.541
C03136=1116.572,414.617,-93.636,-176.604,11.771,149.539
C03137=1116.574,414.370,-93.597,-176.605,11.765,149.538
C03138=1116.576,414.123,-93.558,-176.606,11.760,149.537
C03139=1116.578,413.876,-93.518,-176.607,11.754,149.536
C03140=1116.581,413.630,-93.480,-176.608,11.748,149.534
C03141=1116.584,413.383,-93.440,-176.609,11.742,149.533
C03142=1116.588,413.136,-93.400,-176.610,11.737,149.532
C03143=1116.591,412.889,-93.361,-176.612,11.731,149.531
C03144=1116.595,412.642,-93.322,-176.612,11.725,149.529
C03145=1116.598,412.395,-93.283,-176.614,11.720,149.528
C03146=1116.602,412.148,-93.243,-176.615,11.714,149.527
C03147=1116.606,411.901,-93.204,-176.616,11.709,149.526
C03148=1116.609,411.655,-93.164,-176.617,11.703,149.525
C03149=1116.613,411.408,-93.125,-176.618,11.698,149.524
C03150=1116.616,411.161,-93.086,-176.619,11.693,149.523
C03151=1116.620,410.914,-93.046,-176.621,11.688,149.522
C03152=1116.623,410.667,-93.007,-176.622,11.682,149.520
C03153=1116.627,410.420,-92.968,-176.623,11.677,149.519
C03154=1116.631,410.173,-92.929,-176.624,11.672,149.518
C03155=1116.634,409.926,-92.889,-176.625,11.667,149.517
C03156=1116.637,409.680,-92.851,-176.627,11.661,149.516
C03157=1116.641,409.433,-92.811,-176.628,11.657,149.515
C03158=1116.644,409.186,-92.772,-176.629,11.651,149.514
C03159=1116.648,408.939,-92.733,-176.630,11.646,149.513
C03160=1116.652,408.692,-92.694,-176.631,11.642,149.512
C03161=1116.655,408.445,-92.654,-176.633,11.636,149.511
C03162=1116.659,408.198,-92.615,-176.634,11.632,149.510
C03163=1116.662,407.951,-92.577,-176.635,11.627,149.509
C03164=1116.665,407.704,-92.537,-176.637,11.621,149.508
C03165=1116.670,407.458,-92.498,-176.638,11.617,149.508
C03166=1116.673,407.211,-92.459,-176.640,11.612,149.507
C03167=1116.677,406.964,-92.420,-176.641,11.608,149.506
C03168=1116.680,406.717,-92.382,-176.642,11.602,149.505
C03169=1116.684,406.470,-92.343,-176.643,11.598,149.504
C03170=1116.687,406.223,-92.303,-176.645,11.593,149.503
C03171=1116.691,405.976,-92.264,-176.646,11.589,149.502
C03172=1116.695,405.729,-92.225,-176.648,11.585,149.501
C03173=1116.697,405.482,-92.186,-176.650,11.580,149.501
C03174=1116.701,405.235,-92.148,-176.651,11.575,149.500
C03175=1116.706,404.989,-92.109,-176.653,11.570,149.499
C03176=1116.709,404.742,-92.070,-176.654,11.566,149.498
C03177=1116.712,404.495,-92.031,-176.655,11.562,149.497
C03178=1116.716,404.247,-91.992,-176.657,11.557,149.497
C03179=1116.720,404.000,-91.953,-176.658,11.553,149.496
C03180=1116.723,403.754,-91.915,-176.660,11.549,149.495
C03181=1116.726,403.542,-91.881,-176.661,11.545,149.494
C03182=1116.729,403.330,-91.848,-176.662,11.542,149.494
C03183=1116.732,403.119,-91.815,-176.664,11.538,149.493
C03184=1116.735,402.907,-91.781,-176.665,11.534,149.493
C03185=1116.738,402.695,-91.748,-176.666,11.531,149.492
C03186=1116.742,402.484,-91.715,-176.668,11.527,149.492
C03187=1116.745,402.273,-91.682,-176.669,11.524,149.491
C03188=1116.748,402.061,-91.649,-176.671,11.520,149.490
C03189=1116.751,401.814,-91.610,-176.672,11.516,149.490
C03190=1116.755,401.567,-91.571,-176.674,11.512,149.489
C03191=1116.758,401.320,-91.533,-176.675,11.508,149.489
C03192=1116.762,401.072,-91.494,-176.678,11.504,149.488
C03193=1116.766,400.826,-91.456,-176.679,11.500,149.487
C03194=1116.769,400.579,-91.417,-176.681,11.496,149.487
C03195=1116.773,400.332,-91.378,-176.682,11.492,149.486
C03196=1116.776,400.085,-91.339,-176.684,11.488,149.485
C03197=1116.781,399.838,-91.301,-176.686,11.484,149.485
C03198=1116.784,399.591,-91.262,-176.688,11.481,149.484
C03199=1116.787,399.344,-91.224,-176.689,11.477,149.484
C03200=1116.791,399.097,-91.185,-176.691,11.473,149.483
C03201=1116.794,398.850,-91.147,-176.693,11.469,149.483
C03202=1116.798,398.604,-91.108,-176.694,11.465,149.482
C03203=1116.802,398.356,-91.070,-176.697,11.462,149.482
C03204=1116.805,398.109,-91.032,-176.698,11.458,149.481
C03205=1116.810,397.862,-90.993,-176.700,11.454,149.481
C03206=1116.813,397.615,-90.955,-176.702,11.451,149.480
C03207=1116.816,397.368,-90.915,-176.703,11.448,149.480
C03208=1116.820,397.121,-90.877,-176.705,11.444,149.479
C03209=1116.824,396.874,-90.839,-176.707,11.441,149.479
C03210=1116.827,396.627,-90.801,-176.709,11.437,149.479
C03211=1116.831,396.380,-90.762,-176.711,11.434,149.478
C03212=1116.835,396.133,-90.725,-176.713,11.430,149.478
C03213=1116.838,395.886,-90.685,-176.714,11.427,149.477
C03214=1116.842,395.639,-90.647,-176.717,11.424,149.477
C03215=1116.846,395.391,-90.609,-176.719,11.420,149.477
C03216=1116.849,395.145,-90.571,-176.721,11.417,149.476
C03217=1116.853,394.898,-90.532,-176.723,11.413,149.476
C03218=1116.856,394.651,-90.494,-176.724,11.411,149.475
C03219=1116.861,394.404,-90.456,-176.726,11.407,149.475
C03220=1116.864,394.157,-90.417,-176.729,11.404,149.475
C03221=1116.867,393.910,-90.379,-176.730,11.401,149.474
C03222=1116.871,393.663,-90.341,-176.732,11.397,149.474
C03223=1116.874,393.416,-90.303,-176.734,11.394,149.474
C03224=1116.879,393.169,-90.265,-176.736,11.392,149.474
C03225=1116.882,392.922,-90.226,-176.738,11.388,149.473
C03226=1116.886,392.675,-90.188,-176.740,11.385,149.473
C03227=1116.890,392.428,-90.150,-176.742,11.382,149.473
C03228=1116.893,392.181,-90.112,-176.744,11.379,149.472
C03229=1116.897,391.933,-90.074,-176.746,11.376,149.472
C03230=1116.900,391.687,-90.036,-176.748,11.373,149.472
C03231=1116.904,391.439,-89.998,-176.751,11.370,149.472
C03232=1116.907,391.192,-89.959,-176.752,11.367,149.471
C03233=1116.911,390.946,-89.921,-176.755,11.364,149.471
C03234=1116.914,390.698,-89.884,-176.757,11.362,149.471
C03235=1116.919,390.452,-89.845,-176.759,11.359,149.471
C03236=1116.922,390.204,-89.807,-176.761,11.356,149.470
C03237=1116.925,389.992,-89.775,-176.762,11.353,149.470
C03238=1116.928,389.781,-89.742,-176.764,11.351,149.470
C03239=1116.932,389.569,-89.710,-176.766,11.349,149.470
C03240=1116.934,389.358,-89.677,-176.768,11.346,149.470
C03241=1116.938,389.145,-89.645,-176.770,11.344,149.470
C03242=1116.941,388.933,-89.613,-176.772,11.342,149.470
C03243=1116.944,388.721,-89.579,-176.774,11.339,149.469
C03244=1116.947,388.510,-89.548,-176.776,11.337,149.469
C03245=1116.951,388.263,-89.509,-176.777,11.335,149.469
C03246=1116.955,388.016,-89.472,-176.780,11.331,149.469
C03247=1116.958,387.769,-89.434,-176.782,11.329,149.469
C03248=1116.961,387.521,-89.396,-176.784,11.327,149.469
C03249=1116.966,387.275,-89.358,-176.787,11.324,149.469
C03250=1116.969,387.027,-89.320,-176.789,11.322,149.469
C03251=1116.973,386.781,-89.282,-176.791,11.320,149.469
C03252=1116.976,386.533,-89.244,-176.793,11.316,149.469
C03253=1116.981,386.286,-89.207,-176.796,11.314,149.469
C03254=1116.984,386.039,-89.169,-176.797,11.312,149.468
C03255=1116.988,385.792,-89.131,-176.800,11.309,149.468
C03256=1116.991,385.545,-89.093,-176.802,11.307,149.468
C03257=1116.995,385.298,-89.056,-176.804,11.305,149.468
C03258=1116.999,385.051,-89.017,-176.807,11.302,149.468
C03259=1117.003,384.804,-88.980,-176.809,11.300,149.468
C03260=1117.006,384.556,-88.942,-176.811,11.298,149.468
C03261=1117.010,384.310,-88.905,-176.813,11.295,149.468
C03262=1117.013,384.062,-88.867,-176.816,11.293,149.468
C03263=1117.017,383.815,-88.830,-176.819,11.290,149.468
C03264=1117.021,383.568,-88.791,-176.821,11.288,149.468
C03265=1117.025,383.321,-88.754,-176.823,11.286,149.468
C03266=1117.028,383.074,-88.716,-176.826,11.283,149.468
C03267=1117.032,382.827,-88.679,-176.829,11.281,149.469
C03268=1117.035,382.579,-88.641,-176.832,11.278,149.469
C03269=1117.039,382.333,-88.603,-176.835,11.276,149.469
C03270=1117.042,382.085,-88.566,-176.838,11.273,149.469
C03271=1117.046,381.838,-88.529,-176.842,11.270,149.469
C03272=1117.050,381.591,-88.490,-176.845,11.268,149.469
C03273=1117.054,381.344,-88.453,-176.848,11.265,149.469
C03274=1117.058,381.097,-88.416,-176.851,11.263,149.469
C03275=1117.061,380.849,-88.378,-176.854,11.260,149.469
C03276=1117.065,380.603,-88.341,-176.857,11.257,149.470
C03277=1117.069,380.355,-88.304,-176.860,11.254,149.470
C03278=1117.073,380.108,-88.266,-176.864,11.252,149.470
C03279=1117.077,379.861,-88.229,-176.867,11.250,149.470
C03280=1117.080,379.614,-88.191,-176.870,11.247,149.470
C03281=1117.084,379.366,-88.154,-176.873,11.244,149.470
C03282=1117.087,379.119,-88.117,-176.876,11.242,149.470
C03283=1117.091,378.872,-88.080,-176.879,11.239,149.470
C03284=1117.095,378.625,-88.042,-176.882,11.237,149.471
C03285=1117.098,378.377,-88.005,-176.885,11.235,149.471
C03286=1117.102,378.131,-87.967,-176.888,11.232,149.471
C03287=1117.106,377.884,-87.930,-176.891,11.229,149.471
C03288=1117.110,377.636,-87.893,-176.895,11.227,149.471
C03289=1117.114,377.389,-87.856,-176.898,11.224,149.471
C03290=1117.118,377.142,-87.819,-176.901,11.222,149.472
C03291=1117.121,376.895,-87.781,-176.905,11.219,149.472
C03292=1117.125,376.648,-87.744,-176.907,11.217,149.472
C03293=1117.128,376.436,-87.712,-176.910,11.215,149.472
C03294=1117.131,376.224,-87.680,-176.913,11.213,149.472
C03295=1117.134,376.012,-87.649,-176.916,11.210,149.472
C03296=1117.137,375.800,-87.617,-176.918,11.209,149.473
C03297=1117.141,375.588,-87.585,-176.921,11.206,149.473
C03298=1117.144,375.376,-87.553,-176.924,11.204,149.473
C03299=1117.147,375.164,-87.522,-176.927,11.203,149.473
C03300=1117.150,374.952,-87.490,-176.929,11.200,149.473
C03301=1117.154,374.705,-87.453,-176.933,11.197,149.473
C03302=1117.158,374.458,-87.416,-176.936,11.195,149.474
C03303=1117.161,374.210,-87.378,-176.939,11.192,149.474
C03304=1117.166,373.963,-87.341,-176.942,11.191,149.474
C03305=1117.169,373.716,-87.305,-176.945,11.188,149.474
C03306=1117.173,373.469,-87.268,-176.949,11.186,149.474
C03307=1117.176,373.221,-87.231,-176.952,11.183,149.475
C03308=1117.180,372.975,-87.194,-176.955,11.181,149.475
C03309=1117.184,372.727,-87.157,-176.959,11.178,149.475
C03310=1117.188,372.481,-87.120,-176.962,11.176,149.475
C03311=1117.191,372.233,-87.083,-176.965,11.173,149.475
C03312=1117.195,371.985,-87.046,-176.968,11.171,149.476
C03313=1117.199,371.738,-87.009,-176.972,11.168,149.476
C03314=1117.203,371.491,-86.973,-176.975,11.166,149.476
C03315=1117.206,371.243,-86.936,-176.978,11.163,149.476
C03316=1117.210,370.996,-86.899,-176.982,11.161,149.476
C03317=1117.214,370.749,-86.863,-176.984,11.159,149.477
C03318=1117.218,370.502,-86.826,-176.988,11.157,149.477
C03319=1117.222,370.255,-86.789,-176.991,11.154,149.477
C03320=1117.225,370.007,-86.753,-176.994,11.152,149.477
C03321=1117.229,369.760,-86.716,-176.997,11.149,149.477
C03322=1117.233,369.513,-86.679,-177.001,11.147,149.478
C03323=1117.236,369.266,-86.643,-177.004,11.145,149.478
C03324=1117.240,369.019,-86.606,-177.008,11.142,149.478
C03325=1117.244,368.770,-86.569,-177.011,11.140,149.478
C03326=1117.247,368.524,-86.533,-177.014,11.137,149.479
C03327=1117.252,368.276,-86.496,-177.018,11.135,149.479
C03328=1117.256,368.029,-86.459,-177.021,11.132,149.479
C03329=1117.259,367.782,-86.423,-177.024,11.130,149.479
C03330=1117.263,367.535,-86.386,-177.028,11.127,149.480
C03331=1117.267,367.288,-86.351,-177.031,11.125,149.480
C03332=1117.270,367.040,-86.313,-177.034,11.123,149.480
C03333=1117.274,366.793,-86.276,-177.037,11.121,149.480
C03334=1117.278,366.546,-86.240,-177.041,11.119,149.481
C03335=1117.282,366.298,-86.204,-177.044,11.116,149.481
C03336=1117.285,366.051,-86.168,-177.047,11.114,149.481
C03337=1117.290,365.804,-86.131,-177.051,11.111,149.481
C03338=1117.293,365.556,-86.095,-177.054,11.109,149.482
C03339=1117.297,365.309,-86.059,-177.057,11.106,149.482
C03340=1117.301,365.062,-86.022,-177.061,11.104,149.482
C03341=1117.305,364.814,-85.986,-177.064,11.102,149.482
C03342=1117.308,364.568,-85.950,-177.068,11.099,149.483
C03343=1117.312,364.319,-85.913,-177.071,11.097,149.483
C03344=1117.316,364.072,-85.877,-177.074,11.094,149.483
C03345=1117.320,363.825,-85.840,-177.078,11.092,149.483
C03346=1117.323,363.577,-85.805,-177.081,11.089,149.484
C03347=1117.327,363.330,-85.768,-177.085,11.087,149.484
C03348=1117.331,363.083,-85.732,-177.088,11.085,149.484
C03349=1117.335,362.871,-85.701,-177.091,11.083,149.484
C03350=1117.337,362.659,-85.669,-177.093,11.081,149.485
C03351=1117.340,362.447,-85.639,-177.096,11.079,149.485
C03352=1117.344,362.235,-85.608,-177.099,11.077,149.485
C03353=1117.347,362.023,-85.577,-177.102,11.075,149.485
C03354=1117.351,361.811,-85.546,-177.105,11.073,149.485
C03355=1117.354,361.599,-85.515,-177.108,11.070,149.486
C03356=1117.357,361.386,-85.484,-177.111,11.069,149.486
C03357=1117.361,361.139,-85.448,-177.114,11.066,149.486
C03358=1117.364,360.892,-85.412,-177.117,11.064,149.486
C03359=1117.368,360.644,-85.376,-177.121,11.062,149.487
C03360=1117.372,360.397,-85.340,-177.124,11.059,149.487
C03361=1117.376,360.149,-85.304,-177.128,11.057,149.487
C03362=1117.380,359.902,-85.268,-177.131,11.054,149.487
C03363=1117.384,359.655,-85.232,-177.134,11.052,149.488
C03364=1117.387,359.407,-85.196,-177.138,11.050,149.488
C03365=1117.391,359.160,-85.160,-177.141,11.047,149.488
C03366=1117.394,358.913,-85.124,-177.145,11.045,149.488
C03367=1117.399,358.665,-85.088,-177.148,11.042,149.489
C03368=1117.403,358.418,-85.053,-177.152,11.040,149.489
C03369=1117.407,358.171,-85.017,-177.155,11.038,149.489
C03370=1117.410,357.924,-84.981,-177.158,11.035,149.489
C03371=1117.414,357.676,-84.945,-177.162,11.033,149.490
C03372=1117.418,357.429,-84.909,-177.165,11.030,149.490
C03373=1117.422,357.181,-84.874,-177.169,11.028,149.490
C03374=1117.425,356.934,-84.838,-177.172,11.026,149.491
C03375=1117.430,356.686,-84.802,-177.175,11.023,149.491
C03376=1117.433,356.439,-84.766,-177.179,11.021,149.491
C03377=1117.437,356.191,-84.730,-177.182,11.018,149.491
C03378=1117.440,355.944,-84.695,-177.186,11.016,149.492
C03379=1117.445,355.697,-84.660,-177.189,11.014,149.492
C03380=1117.448,355.450,-84.624,-177.192,11.011,149.492
C03381=1117.453,355.202,-84.588,-177.196,11.009,149.492
C03382=1117.456,354.954,-84.552,-177.199,11.005,149.492
C03383=1117.460,354.707,-84.517,-177.203,11.003,149.493
C03384=1117.464,354.459,-84.481,-177.206,11.001,149.493
C03385=1117.467,354.212,-84.446,-177.210,10.998,149.493
C03386=1117.472,353.965,-84.411,-177.213,10.996,149.494
C03387=1117.475,353.718,-84.375,-177.216,10.993,149.494
C03388=1117.479,353.470,-84.339,-177.220,10.991,149.494
C03389=1117.483,353.223,-84.304,-177.223,10.988,149.494
C03390=1117.486,352.975,-84.268,-177.226,10.986,149.494
C03391=1117.491,352.727,-84.232,-177.230,10.984,149.495
C03392=1117.495,352.480,-84.197,-177.233,10.981,149.495
C03393=1117.499,352.232,-84.162,-177.237,10.978,149.495
C03394=1117.503,351.985,-84.127,-177.241,10.976,149.495
C03395=1117.506,351.737,-84.091,-177.244,10.973,149.496
C03396=1117.510,351.490,-84.056,-177.247,10.971,149.496
C03397=1117.514,351.243,-84.020,-177.250,10.968,149.496
C03398=1117.518,350.995,-83.985,-177.254,10.966,149.496
C03399=1117.522,350.747,-83.950,-177.257,10.963,149.497
C03400=1117.526,350.500,-83.914,-177.261,10.961,149.497
C03401=1117.530,350.253,-83.879,-177.265,10.958,149.497
C03402=1117.533,350.006,-83.844,-177.268,10.956,149.497
C03403=1117.537,349.757,-83.809,-177.271,10.953,149.498
C03404=1117.542,349.511,-83.774,-177.275,10.951,149.498
C03405=1117.544,349.298,-83.744,-177.277,10.949,149.498
C03406=1117.547,349.086,-83.713,-177.280,10.946,149.498
C03407=1117.551,348.873,-83.683,-177.283,10.945,149.498
C03408=1117.554,348.661,-83.654,-177.286,10.942,149.498
C03409=1117.558,348.449,-83.623,-177.289,10.940,149.499
C03410=1117.561,348.237,-83.593,-177.291,10.938,149.499
C03411=1117.564,348.025,-83.564,-177.294,10.936,149.499
C03412=1117.568,347.813,-83.533,-177.296,10.934,149.499
C03413=1117.572,347.565,-83.498,-177.300,10.931,149.499
C03414=1117.575,347.318,-83.463,-177.303,10.929,149.500
C03415=1117.579,347.071,-83.428,-177.306,10.926,149.500
C03416=1117.583,346.823,-83.393,-177.310,10.924,149.500
C03417=1117.587,346.575,-83.357,-177.313,10.921,149.500
C03418=1117.591,346.328,-83.323,-177.316,10.919,149.500
C03419=1117.595,346.080,-83.287,-177.319,10.917,149.501
C03420=1117.599,345.832,-83.252,-177.322,10.914,149.501
C03421=1117.603,345.586,-83.218,-177.325,10.912,149.501
C03422=1117.607,345.337,-83.183,-177.329,10.909,149.501
C03423=1117.611,345.089,-83.148,-177.332,10.907,149.501
C03424=1117.615,344.843,-83.113,-177.335,10.904,149.502
C03425=1117.619,344.594,-83.078,-177.338,10.902,149.502
C03426=1117.622,344.348,-83.044,-177.341,10.899,149.502
C03427=1117.626,344.100,-83.009,-177.345,10.897,149.502
C03428=1117.630,343.852,-82.974,-177.348,10.894,149.502
C03429=1117.634,343.605,-82.939,-177.351,10.892,149.503
C03430=1117.638,343.357,-82.904,-177.354,10.889,149.503
C03431=1117.642,343.110,-82.870,-177.358,10.887,149.503
C03432=1117.646,342.862,-82.834,-177.360,10.885,149.503
C03433=1117.649,342.614,-82.800,-177.364,10.882,149.503
C03434=1117.654,342.367,-82.766,-177.367,10.880,149.504
C03435=1117.657,342.119,-82.730,-177.370,10.877,149.504
C03436=1117.662,341.872,-82.696,-177.373,10.875,149.504
C03437=1117.665,341.624,-82.662,-177.376,10.872,149.504
C03438=1117.670,341.377,-82.627,-177.380,10.870,149.504
C03439=1117.673,341.129,-82.592,-177.383,10.867,149.505
C03440=1117.677,340.882,-82.558,-177.386,10.865,149.505
C03441=1117.681,340.634,-82.523,-177.389,10.862,149.505
C03442=1117.686,340.387,-82.488,-177.393,10.860,149.505
C03443=1117.689,340.139,-82.454,-177.396,10.857,149.505
C03444=1117.694,339.891,-82.420,-177.399,10.855,149.506
C03445=1117.697,339.644,-82.385,-177.402,10.853,149.506
C03446=1117.701,339.397,-82.350,-177.405,10.850,149.506
C03447=1117.705,339.149,-82.315,-177.408,10.848,149.506
C03448=1117.709,338.902,-82.282,-177.411,10.845,149.506
C03449=1117.713,338.653,-82.247,-177.414,10.843,149.506
C03450=1117.717,338.406,-82.213,-177.418,10.840,149.507
C03451=1117.721,338.158,-82.178,-177.421,10.838,149.507
C03452=1117.725,337.911,-82.144,-177.424,10.835,149.507
C03453=1117.728,337.663,-82.109,-177.427,10.833,149.507
C03454=1117.733,337.416,-82.075,-177.431,10.830,149.507
C03455=1117.736,337.168,-82.041,-177.434,10.828,149.508
C03456=1117.741,336.920,-82.006,-177.437,10.825,149.508
C03457=1117.744,336.672,-81.972,-177.440,10.822,149.508
C03458=1117.748,336.425,-81.938,-177.443,10.821,149.508
C03459=1117.752,336.178,-81.904,-177.446,10.818,149.508
C03460=1117.756,335.930,-81.869,-177.449,10.816,149.509
C03461=1117.759,335.717,-81.840,-177.452,10.813,149.509
C03462=1117.762,335.505,-81.811,-177.455,10.811,149.509
C03463=1117.766,335.293,-81.781,-177.457,10.809,149.509
C03464=1117.770,335.081,-81.753,-177.461,10.807,149.509
C03465=1117.773,334.868,-81.723,-177.463,10.805,149.509
C03466=1117.776,334.656,-81.693,-177.466,10.802,149.510
C03467=1117.780,334.443,-81.665,-177.469,10.800,149.510
C03468=1117.783,334.231,-81.635,-177.471,10.799,149.510
C03469=1117.788,333.984,-81.601,-177.474,10.796,149.510
C03470=1117.791,333.736,-81.566,-177.477,10.793,149.510
C03471=1117.795,333.488,-81.533,-177.481,10.791,149.511
C03472=1117.799,333.240,-81.498,-177.484,10.789,149.511
C03473=1117.803,332.993,-81.464,-177.487,10.786,149.511
C03474=1117.807,332.745,-81.430,-177.490,10.783,149.511
C03475=1117.811,332.497,-81.396,-177.494,10.781,149.511
C03476=1117.815,332.250,-81.363,-177.497,10.778,149.511
C03477=1117.818,332.003,-81.329,-177.500,10.776,149.512
C03478=1117.823,331.754,-81.295,-177.503,10.774,149.512
C03479=1117.827,331.507,-81.261,-177.506,10.772,149.512
C03480=1117.830,331.260,-81.227,-177.509,10.769,149.512
C03481=1117.835,331.011,-81.193,-177.512,10.766,149.512
C03482=1117.838,330.764,-81.159,-177.516,10.764,149.513
C03483=1117.842,330.517,-81.125,-177.518,10.761,149.513
C03484=1117.847,330.268,-81.091,-177.522,10.759,149.513
C03485=1117.850,330.021,-81.057,-177.525,10.756,149.513
C03486=1117.855,329.773,-81.024,-177.528,10.754,149.514
C03487=1117.858,329.525,-80.990,-177.531,10.751,149.514
C03488=1117.862,329.278,-80.956,-177.535,10.749,149.514
C03489=1117.867,329.030,-80.922,-177.538,10.746,149.514
C03490=1117.871,328.783,-80.889,-177.541,10.743,149.514
C03491=1117.874,328.535,-80.855,-177.544,10.742,149.514
C03492=1117.878,328.287,-80.821,-177.547,10.739,149.515
C03493=1117.883,328.040,-80.787,-177.550,10.736,149.515
C03494=1117.887,327.792,-80.754,-177.553,10.734,149.515
C03495=1117.890,327.544,-80.720,-177.556,10.732,149.515
C03496=1117.894,327.296,-80.686,-177.559,10.729,149.515
C03497=1117.898,327.049,-80.653,-177.563,10.726,149.515
C03498=1117.902,326.801,-80.619,-177.566,10.724,149.516
C03499=1117.906,326.553,-80.586,-177.569,10.721,149.516
C03500=1117.910,326.306,-80.551,-177.572,10.719,149.516
C03501=1117.914,326.058,-80.518,-177.576,10.716,149.516
C03502=1117.918,325.810,-80.485,-177.579,10.714,149.517
C03503=1117.922,325.562,-80.451,-177.581,10.712,149.517
C03504=1117.926,325.315,-80.418,-177.585,10.709,149.517
C03505=1117.930,325.067,-80.385,-177.588,10.707,149.517
C03506=1117.934,324.819,-80.351,-177.591,10.704,149.517
C03507=1117.938,324.572,-80.318,-177.594,10.702,149.517
C03508=1117.941,324.324,-80.284,-177.597,10.699,149.518
C03509=1117.946,324.076,-80.251,-177.600,10.696,149.518
C03510=1117.950,323.828,-80.218,-177.604,10.694,149.518
C03511=1117.954,323.581,-80.184,-177.607,10.691,149.518
C03512=1117.958,323.333,-80.151,-177.610,10.689,149.518
C03513=1117.962,323.086,-80.118,-177.613,10.686,149.519
C03514=1117.965,322.837,-80.084,-177.616,10.683,149.519
C03515=1117.970,322.589,-80.051,-177.619,10.682,149.519
C03516=1117.974,322.342,-80.018,-177.622,10.679,149.519
C03517=1117.977,322.129,-79.989,-177.625,10.677,149.519
C03518=1117.981,321.917,-79.961,-177.628,10.675,149.519
C03519=1117.984,321.704,-79.932,-177.630,10.673,149.520
C03520=1117.988,321.491,-79.903,-177.633,10.670,149.520
C03521=1117.991,321.279,-79.875,-177.636,10.668,149.520
C03522=1117.995,321.066,-79.846,-177.639,10.666,149.520
C03523=1117.997,320.854,-79.818,-177.641,10.664,149.520
C03524=1118.001,320.642,-79.789,-177.644,10.662,149.520
C03525=1118.006,320.394,-79.756,-177.647,10.660,149.521
C03526=1118.010,320.146,-79.723,-177.650,10.657,149.521
C03527=1118.012,319.898,-79.690,-177.653,10.654,149.521
C03528=1118.017,319.650,-79.657,-177.656,10.652,149.521
C03529=1118.021,319.403,-79.624,-177.659,10.649,149.521
C03530=1118.025,319.155,-79.591,-177.663,10.647,149.521
C03531=1118.029,318.907,-79.558,-177.666,10.644,149.522
C03532=1118.033,318.660,-79.524,-177.669,10.641,149.522
C03533=1118.037,318.412,-79.491,-177.672,10.639,149.522
C03534=1118.041,318.164,-79.459,-177.675,10.637,149.522
C03535=1118.045,317.917,-79.426,-177.678,10.635,149.522
C03536=1118.049,317.669,-79.392,-177.681,10.632,149.522
C03537=1118.053,317.421,-79.359,-177.684,10.629,149.523
C03538=1118.058,317.173,-79.327,-177.688,10.627,149.523
C03539=1118.061,316.925,-79.294,-177.690,10.624,149.523
C03540=1118.065,316.678,-79.261,-177.694,10.622,149.523
C03541=1118.069,316.430,-79.228,-177.697,10.619,149.523
C03542=1118.073,316.182,-79.195,-177.700,10.617,149.524
C03543=1118.077,315.934,-79.163,-177.703,10.614,149.524
C03544=1118.081,315.686,-79.130,-177.706,10.611,149.524
C03545=1118.085,315.439,-79.097,-177.710,10.609,149.524
C03546=1118.090,315.191,-79.064,-177.712,10.607,149.524
C03547=1118.093,314.943,-79.032,-177.715,10.604,149.525
C03548=1118.097,314.695,-78.999,-177.719,10.602,149.525
C03549=1118.101,314.447,-78.965,-177.721,10.599,149.525
C03550=1118.105,314.199,-78.934,-177.725,10.597,149.525
C03551=1118.109,313.952,-78.900,-177.728,10.594,149.525
C03552=1118.113,313.704,-78.867,-177.731,10.592,149.525
C03553=1118.117,313.456,-78.835,-177.734,10.589,149.526
C03554=1118.121,313.208,-78.802,-177.737,10.586,149.526
C03555=1118.126,312.960,-78.770,-177.741,10.584,149.526
C03556=1118.129,312.712,-78.737,-177.744,10.581,149.526
C03557=1118.133,312.465,-78.704,-177.747,10.579,149.526
C03558=1118.138,312.216,-78.672,-177.749,10.577,149.526
C03559=1118.141,311.969,-78.639,-177.753,10.574,149.527
C03560=1118.146,311.721,-78.607,-177.756,10.572,149.527
C03561=1118.149,311.473,-78.574,-177.759,10.569,149.527
C03562=1118.154,311.226,-78.542,-177.762,10.567,149.527
C03563=1118.158,310.978,-78.509,-177.765,10.564,149.527
C03564=1118.162,310.730,-78.477,-177.768,10.561,149.528
C03565=1118.166,310.482,-78.444,-177.771,10.559,149.528
C03566=1118.170,310.234,-78.412,-177.775,10.556,149.528
C03567=1118.174,309.986,-78.379,-177.778,10.554,149.528
C03568=1118.178,309.738,-78.347,-177.781,10.551,149.528
C03569=1118.182,309.490,-78.315,-177.784,10.549,149.529
C03570=1118.186,309.243,-78.282,-177.787,10.547,149.529
C03571=1118.190,308.995,-78.250,-177.790,10.544,149.529
C03572=1118.194,308.747,-78.218,-177.793,10.541,149.529
C03573=1118.198,308.534,-78.189,-177.796,10.539,149.529
C03574=1118.201,308.321,-78.162,-177.798,10.537,149.529
C03575=1118.205,308.109,-78.135,-177.801,10.535,149.529
C03576=1118.208,307.896,-78.106,-177.804,10.533,149.530
C03577=1118.212,307.684,-78.079,-177.806,10.531,149.530
C03578=1118.215,307.470,-78.051,-177.809,10.529,149.530
C03579=1118.219,307.259,-78.023,-177.812,10.526,149.530
C03580=1118.222,307.045,-77.996,-177.814,10.524,149.530
C03581=1118.227,306.798,-77.964,-177.818,10.522,149.531
C03582=1118.231,306.550,-77.932,-177.821,10.519,149.531
C03583=1118.234,306.302,-77.900,-177.824,10.516,149.531
C03584=1118.238,306.054,-77.867,-177.827,10.514,149.531
C03585=1118.242,305.806,-77.835,-177.830,10.511,149.531
C03586=1118.247,305.558,-77.803,-177.832,10.509,149.531
C03587=1118.251,305.310,-77.771,-177.836,10.507,149.532
C03588=1118.255,305.062,-77.739,-177.839,10.504,149.532
C03589=1118.259,304.814,-77.707,-177.842,10.502,149.532
C03590=1118.263,304.567,-77.674,-177.845,10.499,149.532
C03591=1118.267,304.319,-77.642,-177.848,10.496,149.532
C03592=1118.271,304.071,-77.610,-177.851,10.494,149.532
C03593=1118.275,303.823,-77.578,-177.855,10.491,149.533
C03594=1118.280,303.575,-77.546,-177.857,10.488,149.533
C03595=1118.284,303.327,-77.514,-177.861,10.486,149.533
C03596=1118.287,303.079,-77.483,-177.864,10.484,149.533
C03597=1118.292,302.832,-77.451,-177.866,10.482,149.533
C03598=1118.296,302.583,-77.419,-177.870,10.479,149.534
C03599=1118.300,302.335,-77.387,-177.873,10.476,149.534
C03600=1118.304,302.088,-77.355,-177.876,10.474,149.534
C03601=1118.309,301.839,-77.323,-177.879,10.471,149.534
C03602=1118.312,301.591,-77.291,-177.882,10.469,149.534
C03603=1118.317,301.344,-77.260,-177.885,10.466,149.534
C03604=1118.320,301.096,-77.228,-177.889,10.464,149.535
C03605=1118.325,300.848,-77.195,-177.891,10.461,149.535
C03606=1118.329,300.600,-77.164,-177.895,10.458,149.535
C03607=1118.333,300.352,-77.133,-177.898,10.456,149.535
C03608=1118.337,300.104,-77.101,-177.900,10.454,149.535
C03609=1118.341,299.856,-77.069,-177.903,10.451,149.535
C03610=1118.345,299.608,-77.037,-177.907,10.449,149.536
C03611=1118.349,299.360,-77.005,-177.910,10.446,149.536
C03612=1118.354,299.113,-76.974,-177.913,10.444,149.536
C03613=1118.358,298.864,-76.942,-177.916,10.441,149.536
C03614=1118.361,298.616,-76.911,-177.919,10.438,149.536
C03615=1118.366,298.369,-76.879,-177.922,10.436,149.536
C03616=1118.370,298.120,-76.847,-177.926,10.433,149.537
C03617=1118.375,297.872,-76.816,-177.928,10.430,149.537
C03618=1118.378,297.624,-76.784,-177.931,10.429,149.537
C03619=1118.382,297.376,-76.752,-177.934,10.426,149.537
C03620=1118.386,297.129,-76.721,-177.937,10.424,149.537
C03621=1118.390,296.880,-76.690,-177.940,10.421,149.538
C03622=1118.395,296.633,-76.658,-177.944,10.418,149.538
C03623=1118.398,296.385,-76.626,-177.947,10.416,149.538
C03624=1118.402,296.136,-76.595,-177.950,10.413,149.538
C03625=1118.407,295.889,-76.564,-177.953,10.410,149.538
C03626=1118.411,295.640,-76.532,-177.956,10.408,149.538
C03627=1118.415,295.393,-76.501,-177.959,10.405,149.539
C03628=1118.419,295.145,-76.469,-177.961,10.403,149.539
C03629=1118.423,294.932,-76.443,-177.965,10.401,149.539
C03630=1118.426,294.719,-76.415,-177.967,10.399,149.539
C03631=1118.429,294.506,-76.388,-177.970,10.396,149.539
C03632=1118.433,294.293,-76.361,-177.972,10.394,149.539
C03633=1118.436,294.081,-76.335,-177.975,10.392,149.540
C03634=1118.440,293.868,-76.308,-177.978,10.390,149.540
C03635=1118.444,293.655,-76.281,-177.980,10.388,149.540
C03636=1118.447,293.442,-76.254,-177.983,10.386,149.540
C03637=1118.452,293.194,-76.223,-177.986,10.383,149.540
C03638=1118.455,292.946,-76.191,-177.989,10.380,149.540
C03639=1118.459,292.698,-76.161,-177.992,10.378,149.541
C03640=1118.463,292.450,-76.130,-177.995,10.375,149.541
C03641=1118.468,292.202,-76.098,-177.998,10.373,149.541
C03642=1118.472,291.954,-76.067,-178.001,10.370,149.541
C03643=1118.476,291.706,-76.036,-178.005,10.368,149.541
C03644=1118.480,291.458,-76.004,-178.007,10.366,149.541
C03645=1118.485,291.210,-75.974,-178.010,10.363,149.542
C03646=1118.488,290.962,-75.942,-178.013,10.360,149.542
C03647=1118.493,290.714,-75.911,-178.017,10.358,149.542
C03648=1118.497,290.466,-75.881,-178.020,10.355,149.542
C03649=1118.501,290.218,-75.849,-178.023,10.353,149.542
